(* CoDeSys 2.3 project: cy_64_Desenzano_geolum_1.pro *)
(* Title: cy-wg-24 - ClevergyAS *)
(* Author: Andrea Laini *)
(* Libraries: mod_com.lib 16.5.13 14:00:50, SerComm.lib 16.5.13 14:00:50, GitHubLocalRepository\FIRMWARE_BUILDING_BLOCKS\LuxBlock\LUX_v2.lib 20.4.16 07:33:55, Serial_Interface_01.lib 22.4.13 12:50:14, WagoLibLed.lib 17.6.13 10:40:56, Modb_l05.lib 13.5.15 10:30:08, SysLibFile.lib 16.5.13 14:00:50, Util.lib 16.5.13 14:00:50, GitHubLocalRepository\FIRMWARE_BUILDING_BLOCKS\AstrBlock\obj_ASTR_v2.lib 20.4.16 07:33:55, SYSLIBCALLBACK.LIB 16.5.13 14:00:50, WAGO-CODESYS-LIBS\OSCAT\oscat_basic_333_pfc_2000.lib 10.4.16 18:08:12, SysLibRtc.lib 16.5.13 14:00:50, SysLibSockets.lib 22.5.14 16:16:32, SysLibEvent.lib 16.5.13 14:00:50, SysLibTime.lib 16.5.13 14:00:48, SysLibPlcCtrl.lib 16.5.13 14:00:50, GitHubLocalRepository\FIRMWARE_BUILDING_BLOCKS\CronoBlocks\crono_pfc2000.lib 20.4.16 07:33:55, SysLibStr.lib 16.5.13 14:00:50, Standard.lib 20.5.14 08:13:26, GitHubLocalRepository\FIRMWARE_BUILDING_BLOCKS\01_Lib_ClevergyUtils\ClevergyUtils_pcf2000.lib 20.4.16 07:33:55, Iecsfc.lib 16.5.13 14:00:50 *)

(* PLC configuration (modules and I/O channels)
VPN_STATUS AT %IX0.0 [BOOLOnX_I] I 1: Digital Input
DI02 AT %IX0.1 [BOOLOnX_I] I 2: Digital Input
COORD_STATUS AT %IX0.2 [BOOLOnX_I] I 3: Digital Input
DI04 AT %IX0.3 [BOOLOnX_I] I 4: Digital Input
Modbus variables [PFC200MODBUS] node 1, in %IB0 out %QB0 {PlcStopBehaviour = 1; FiledbusErrorBehaviour = 1; TcpOperation = 0; TcpPort = 502; TcpTimeout = 600; UdpOperation = 0; UdpPort = 502; RtuOperation = 0; NodeId = 200; ResponseTimeout = 5000; Interface = 0; Baud = 38400; StopBits = 2; Parity = 0; FlowCtrl = 0; PhysInterface = 1}
Modbus-Master [MB_MASTER] node 2, in %IB0 out %QB0
*)

(* Global variable list: Global_Constants *)
VAR_GLOBAL CONSTANT

	Plant_NAME			: STRING :='cySN:64  cyVER:0 - Desenzano lab testing';
	Plant_SN				: DWORD  :=64;	  	(* S/N Impianto di telecontrollo *)
	Plant_SW_VER			: WORD   :=0;		(* Versione SW installata *)

	(* Plant-dependent constants *)
	LATITUDE 										: REAL:=45.660772;
	LONGITUDE										: REAL:=9.652021;
	ASTRO_TWILIGHT_MORNING_MODE					: BYTE:=50;
	ASTRO_TWILIGHT_EVENING_MODE					: BYTE:=50;
	COUNTRY_CODE 									: STRING:='IT';
	MAX_LUXNUM										: WORD := 150;
	MAX_GEOLUMENNODES								: WORD :=MAX_LUXNUM;
	MAX_RETRY_NO_FEEDBACK_GEOLUMEN_NODES			: WORD:=5;
	MAX_RETRY_STATUS_NOT_ALIGNED_GEOLUMEN_NODES       : WORD:=60;

	(* Internal, tech const *)
	MAX_ARRAY_MSG	: BYTE:=250;
	ANALOG			: BOOL:=0;
	DIGITAL			: BOOL:=1;

	(* Filesystem *)
	FilesPath  			: STRING :='/media/sd/';
	MapConf_Path			: STRING :=	'/media/sd/';

	Luxlist_FileName	: STRING :='_LUX_LIST.txt';
	Cfg_FileName		: STRING :='CFG.txt';

	(* Colour Visu *)
	COLOR_RED			: DWORD 	:= 16#2020F0;
	COLOR_YELLOW		: DWORD	:= 16#20F0F0;
	COLOR_GREEN		: DWORD	:= 16#20F020;
	COLOR_GREEN_OFF	 : DWORD	:= 16#108010;

	(* TCP Logger *)
	Logger_SERVER		: STRING:='';
	Logger_IP				: STRING:='192.168.100.3';
	Logger_PORT			: WORD  :=80;
	Logger_GETSTART		: STRING:='GET /cygmsrv/hsgm.ashx?';
	Logger_GETEND		: STRING:='$R$N$R$N';
	Logger_CHECK			: STRING:='True';
	Logger_CRLF			: STRING:='$R$N';
	Logger_DataFile		: STRING:='/media/sd/LOG.DAT';
	Logger_DataFileOld	: STRING:='/media/sd/LOG.BCK';
	Logger_IndexFile	: STRING:='/media/sd/LOG.IDX';
	Logger_ConnRetries	: BYTE:=5;
	Logger_RecoverMsgs	: BYTE:=25;

	(* TCP Remote *)
	Remote_PORT			: WORD  :=10;
	Remote_WELCOME		: STRING:='Connected$R$N';
	Remote_OK			: STRING:='OK$R$N';
	Remote_ERROR		: STRING:='ERROR$R$N';

	(* TCP Sockets *)
	MAX_SEND_TCP_SERVER					 : DWORD:=3000;(*60000*)
	MAX_RECEIVE_TCP_SERVER				 : DWORD:=3000;
	MAX_RECEIVE_TCP_SERVER_SOCKET	 	 : DWORD:=1500;
	MAX_SEND_TCP_CLIENT					 : DWORD:=3000;(*15000*)
	MAX_RECEIVE_TCP_CLIENT				 : DWORD:=1500;
	MAX_RECEIVE_TCP_CLIENT_SOCKET		 : DWORD:=1500;
	MAX_RECEIVE_UDP_SERVER				 : INT  :=1472;
	MAX_RECEIVE_UDP_CLIENT				 : INT  :=1472;
	CONNECT_WATCHDOG_TIME				 : TIME :=t#10s;


END_VAR

(* Global variable list: Global_Retain *)
VAR_GLOBAL RETAIN PERSISTENT

	(* valori retain per i LUX objects*)
	GlobalWorkingtime		: ARRAY [1..MAX_LUXNUM] OF DWORD; (* [sec] Internal working time counter *)
	GlobalPowerOnCycles	: ARRAY [1..MAX_LUXNUM] OF WORD;	(*/DWORD;  *) (* Internal counter of power-on cycles *)
	GlobalEnergyCounter	: ARRAY [1..MAX_LUXNUM] OF WORD; (* DWORD;  *) (* [E-1 kWh] Internal energy counter *)
	GlobalEnergyCounter_t 	: ARRAY [1..MAX_LUXNUM] OF DWORD; (* Temporary energy in E-2*Wsec *)

 	(*Tabella della lista dei lux GEOLUMEN costruita sulla base del file di configurazione*)
	TabListLux : ARRAY [1..MAX_LUXNUM] OF type_TabListLuxGeolumen;

	LuxElement		: ARRAY [1..MAX_LUXNUM] OF obj_LUX;  (* Lista di variabili Lux   *)
	LuxGeolumenChangeFlag : ARRAY [1..MAX_LUXNUM] OF INT;

	(*configurazione degli astro *)
	ASTR_CONFIG   : ARRAY [1..MAX_LUXNUM] OF  type_ASTR_config;

	USE_RETAIN:BOOL:=FALSE;

END_VAR

(* Global variable list: Global_Variables *)
VAR_GLOBAL

	SYS    : typ_SYS;
	Logger : typ_Logger;

	LAMP : LAMP_AL_GENERALE;

	PLC_ID				: STRING:='1' ; (* Identificativo del plc - interno al file cfg.txt  *)

	SyncLogRequest: BOOL:=FALSE;
	TimerLogLux : ARRAY[1..15] OF TON;
	TimerLogLuxSync : ARRAY[1..15] OF TON;
	TimerLogLuxSyncDone : ARRAY[1..15] OF BOOL;
	TimingLuxBase : TIME;
	logRowLux:INT:=0;

	TimerLogAstro : ARRAY[1..15] OF TON;
	TimerLogAstroSync : ARRAY[1..15] OF TON;
	TimerLogAstroSyncDone : ARRAY[1..15] OF BOOL;
	TimingAstroBase : TIME;
	tIndex:INT;
	logRowAstro:INT:=0;

	GeolumenNodeList	:GeolumenNodeList;

	(* Astro crono *)
	ASTR   			: ARRAY [1..MAX_LUXNUM] OF obj_ASTR;
	astroGen : obj_ASTR;
	CronEd : obj_CRON_EDITOR:=(crono_type:='ASTR');

	(*Lux *)
	MsgRecBuffer	: ARRAY[0..MAX_ARRAY_MSG ] OF type_MsgReceive; (*Array contenente i messaggi in arrivo e gestito in modo circolare*)
	KEYON :BOOL;

	DataLuxForVis	: ARRAY [1..MAX_LUXNUM] OF type_DataLuxForVis;	(*ARRAY ordinato contenente i valori Status_Vis e del timer utilizzati per la visualizzazione (PLC_Visualization)*)

	LuxGeolumenNodes : ARRAY [1..MAX_LUXNUM] OF obj_GeolumenNode:=(MAX_RETRY_NO_FEEDBACK:=MAX_RETRY_NO_FEEDBACK_GEOLUMEN_NODES,
															MAX_RETRY_STATUS_NOT_ALIGNED:=MAX_RETRY_STATUS_NOT_ALIGNED_GEOLUMEN_NODES);

	LuxGeolumenNodesAlignFlags : ARRAY [1..MAX_LUXNUM] OF BOOL:=FALSE;

	(*Geolumen rs232 dependent*)
	COM0:SERIAL_INTERFACE := (xOPEN_COM_PORT := TRUE, bCOM_PORT_NR  := 0, cbsBYTESIZE := BS_8,
							cbBAUDRATE := BAUD_38400, cpPARITY := PARITY_NO, csSTOPBITS := STOPBITS_1, cfFLOW_CONTROL := NO_FLOW_CONTROL);
	ReceiveBuffer, ReceiveBufferTrash	:typRing_Buffer;
	xCoupledAll		:BOOL;
	obj_GeolumenCoordinator:obj_GeolumenCoordinator;
	LuxGeolumenDiagnostics:LuxGeolumenDiagnostics;
	SendDataQueue:SendDataQueue;

END_VAR

(* Data type in System *)
TYPE en_MsgType :
(
	COMPLETED:=0, (*Il messaggio è stato elaborato*)
	REQAUTH0:= 1,  (*Richiesta in corso a cui rispondere*)
	REQAUTH1:=2,  (*Nodo già acquisito in rete*)
	DATAREC:=3,
	ECHO:=4,
	NODE_DELETED:=5
);
END_TYPE

(* Data type in System *)
TYPE en_StartingState :
(
	NOT_AUTHORISE  := 0,
	READ_NODE
);
END_TYPE

(* Data type *)
TYPE type_ASTR_config :
STRUCT
	id:DWORD;
	twilightMorningMode:BYTE;
	twilightEveningMode:BYTE;
	preSunrise:BYTE;
	postSunrise:BYTE;
	preSunset:BYTE;
	postSunset:BYTE;
END_STRUCT
END_TYPE

(* Data type in DT_LUX_GEOLUMEN *)
TYPE type_LuxGeolumenStatus :
STRUCT
	ID_Geolumen: DWORD;
	DimmValue_0 : WORD;
	DimmValue_1 : WORD;
	DimmValue_2 : WORD;
END_STRUCT
END_TYPE

(* Data type in System *)
TYPE type_MsgReceive :
STRUCT
	Msg		:STRING (255);
	MsgType	: en_MsgType; (*Indica il tipo di messaggio STS0, STS1,...*)
	dwMacAdd	: DWORD;

END_STRUCT
END_TYPE

(* Data type in DT_LUX_GEOLUMEN *)
(* Struttura utile per la lista dei lux *)

TYPE type_TabListLuxGeolumen :
STRUCT
	LuxNumber	: DWORD;
	LuxID_Geolumen		: DWORD;
	MacAdd	: DWORD;
	MacAddH	: WORD;
	MacAddL	: WORD;
	StMacAdd	: STRING(8);
	xCoupled	: BOOL;
END_STRUCT
END_TYPE

(* POU PLC_PRG, ST *)
PROGRAM PLC_PRG
VAR CONSTANT
	TIME_LUX_LOG_NORMAL:TIME:=T#5m;
	TIME_ASTRO_LOG_NORMAL:TIME:=T#6m30s;
END_VAR
VAR

 	Timer1: TON;  (*Fast controls tick *)
  	Timer2: TON; (* Plant control tick *)
	Timer3: TON; (* Logger timer *)
	Timer4: TON; (* Logger timer *)
	Timer5: TON; (* Logger timer *)


	xOpenPort		: BOOL := TRUE;
	xInitPort			: BOOL;
	xSendActive	: BOOL;
	SendString		: STRING(255) := 'CMD_AUTHORISE=1';
	xStartSend		: BOOL;

(* Application vars *)



	i :INT :=0;
	InitCom: BOOL;
	temp 		: BYTE;
	temp2		: INT;



	LuxCount	: WORD;
	LuxEnInfo	: BOOL;
	ValInCrono	: INT; (* Valore del setpoint del crono *)
	counter		: WORD;


	tmpIndex:INT;



END_VAR
(*
	Network setup:
		IP  = 192.168.100.2 | MSK = 255.255.255.0
		GW	= 192.168.100.1 | DNS = 192.168.100.1
		SNTP = 193.204.114.232 (3600s) ==> 192.168.100.3
*)


(*==============================*)
(*=====    Main control machine    ====*)
(*==============================*)

MainCtrl();

Logger_Proc();

Remote_Proc();
END_PROGRAM
ACTION MainCtrl:
CASE Sys.Status OF

	S_STARTUP:
		(* Load the allowed Geolumen nodes *)
		GeolumenNodeList();
		FOR counter := 1 TO MAX_LUXNUM DO
			LuxElement[counter].DimmingType:=1;
			LuxElement[counter].CTRL_MODE := 2 ; (* TabDefaultLux[counter].Mode; //copio il mode nella tabella delle variabili dei lux 	*)
			LuxElement[counter].CTRL_MODE_backUp := 2;  (* TabDefaultLux[counter].Mode; //salvo il mode di backup per il ripristina modo	*)
		END_FOR

		(* apro la porta seriale *)
		xSendActive:=FALSE;
		COM0((*	bCOM_PORT_NR 	:= 0,
				cbBAUDRATE     	 := BAUD_38400,
			(*	cbBAUDRATE 		:= wBaudRate, *)
				cbsBYTESIZE		:= BS_8,  (*bDataBits,*)
				cpPARITY			:= PARITY_NO, (* bParity,*)
				csSTOPBITS		:= STOPBITS_1,
				cfFLOW_CONTROL	:= NO_FLOW_CONTROL,	(*bFlowControl,			*) *)
				utRECEIVE_BUFFER := ReceiveBuffer,
				ptSEND_BUFFER	:= ADR(SendString),
				xINIT				:=  xInitPort,
		     		xOPEN_COM_PORT 	:= TRUE,	(*xOpenPort,*)
				iBYTES_TO_SEND	:= LEN(SendString)+1,
				xSTART_SEND		:= xSendActive );

		IF COM0.xCOM_PORT_IS_OPEN THEN
			Sys.Status:=S_INIT_RTC;
		END_IF

	S_INIT_RTC:

		(* anzitutto blocco auto-accesso da parte dei nodi*)
		obj_GeolumenCoordinator.blockNodeAutoAdd_direct();

		(* Check RTC and update from network *)
		RTC_Update();
		(* Check time *)
		IF Sys.Time_Year>2000 THEN
			obj_GeolumenCoordinator.updateNetworkTime();
			Sys.Status:=S_INIT_VAR;
		END_IF

	S_INIT_VAR:
		(*ripeto il comando di esclusione di accesso da parte dei nodi, per sicurezza*)
		obj_GeolumenCoordinator.blockNodeAutoAdd();

		(* inizializzo gli astro con eventale stato retain *)
		FOR i:=1 TO max_luxnum DO
			ASTR[i].ID:=ASTR_CONFIG[i].ID;
			ASTR[i].rLatitude:=LATITUDE;
			ASTR[i].rLongitude:=LONGITUDE;
			ASTR[i].countryCode:=COUNTRY_CODE;
			IF(USE_RETAIN=FALSE) THEN
				ASTR[i].twilightEveningMode :=ASTRO_TWILIGHT_EVENING_MODE;
				ASTR[i].twilightMorningMode :=ASTRO_TWILIGHT_MORNING_MODE;
				ASTR_CONFIG[i].preSunrise:=ASTR[i].preSunrise;
				ASTR_CONFIG[i].postSunrise:=ASTR[i].postSunrise;
				ASTR_CONFIG[i].preSunset:=ASTR[i].preSunset;
				ASTR_CONFIG[i].postSunset:=ASTR[i].postSunset;
				ASTR_CONFIG[i].twilightEveningMode:=ASTR[i].twilightEveningMode;
				ASTR_CONFIG[i].twilightMorningMode:=ASTR[i].twilightMorningMode;
			ELSE
				ASTR[i].preSunrise:=ASTR_CONFIG[i].preSunrise;
				ASTR[i].postSunrise:=ASTR_CONFIG[i].postSunrise;
				ASTR[i].preSunset:=ASTR_CONFIG[i].preSunset;
				ASTR[i].postSunset:=ASTR_CONFIG[i].postSunset;
				ASTR[i].twilightEveningMode:=ASTR_CONFIG[i].twilightEveningMode;
				ASTR[i].twilightMorningMode:=ASTR_CONFIG[i].twilightMorningMode;
			END_IF

		END_FOR

		(*chiedo agli eventuali nodi geoluem connesso il loro stato già connessi stato *)
		SendDataQueue(pTxData:=ADR(obj_GeolumenCoordinator.getStatusAllFeedback),ReceiveBufferPtr:=ADR(ReceiveBuffer));
		SendDataQueue.addMessage();
		SendDataQueue();

		Sys.Status:=S_STARTER;

	S_STARTER:
		LogEv(EL_Wrn,EO_SYS,0,1,CONCAT('System_startup_v',WORD_TO_STRING(Plant_SW_VER)));
		Sys.Status:=S_RUNNING;

	S_RUNNING:

		astroGen(ID:=1);

		Timer1(IN:=NOT Timer1.Q,PT:=T#50ms);
		IF Timer1.Q THEN
			(* Update meters *)
			SCA_Proc();
			(* Update system checks *)
			SYS_Proc();
		END_IF

		Timer2(IN:=NOT Timer2.Q,PT:=T#500MS);
		IF Timer2.Q THEN
			(* Read current date/time *)
			RTC_Update();
		END_IF

		obj_GeolumenCoordinator(ReceiveBufferPtr:=ADR(ReceiveBuffer),MsgRecBufferPtr:=ADR(MsgRecBuffer));

		(* Execute Cron Editor commands *)
		CronEd();

		(*Timer4(IN:=NOT Timer4.Q,PT:=T#500ms);
		IF Timer4.Q THEN*)



			FOR LuxCount:=1 TO  MAX_LUXNUM DO

				(*eseguo diagnostica lux*)
				LuxGeolumenDiagnostics();

				IF  LuxElement[LuxCount].ID <> 0  THEN (* esegue scansione dei lux dell'impianto solo se presenti *)

					(* salvo lo stato desiderato corrente del LuxGeolumenNode *)
					LuxGeolumenChangeFlag[LuxCount]:=LuxGeolumenNodes[LuxCount].desideredDimmValue;

					CASE LuxElement[LuxCount].CTRL_MODE OF
						(*
						0:
						1:	 *)
						2:

							IF  ASTR[LuxCount].ID <> 0 THEN
								(* se il mode è settato come cronografo gestisco accensione a orologio *)
								ASTR[LuxCount]( localTime:=Sys.Time_CT_DT,SetPoint=>ValInCrono);
								LuxElement[LuxCount].ValInCronoInLux:=ValInCrono;
							END_IF

					END_CASE

					LuxElement[LuxCount](	LuxAnalogOut => LuxGeolumenNodes[LuxCount].desideredDimmValue,
										WorkingTime:=GlobalWorkingtime[LuxCount],
										PowerOnCycles:=GlobalPowerOnCycles[LuxCount],
										EnergyCounter:=GlobalEnergyCounter[LuxCount],
										EnergyCounter_t:=GlobalEnergyCounter_t[LuxCount],KeyQty:=2);  (*, KeyMode:=KeyTest.KeyMode); *)

					(* aggiorno lo stato desiderato del LUX GeolumenNode*)
					LuxGeolumenNodes[LuxCount].updateDesideredState();
					(* se è diverso dal precedente, invio richiesta modifica stato *)
					IF(LuxGeolumenChangeFlag[LuxCount]<>LuxGeolumenNodes[LuxCount].desideredDimmValue) THEN
						(*invio set*)
						SendDataQueue(pTxData:=ADR(LuxGeolumenNodes[LuxCount].toSendSetString),ReceiveBufferPtr:=ADR(ReceiveBuffer));
						SendDataQueue.addMessage();
						(*invio get*)
						SendDataQueue(pTxData:=ADR(LuxGeolumenNodes[LuxCount].toSendGetString),ReceiveBufferPtr:=ADR(ReceiveBuffer));
						SendDataQueue.addMessage();
						SendDataQueue();
					END_IF

					LuxGeolumenNodes[LuxCount].checkStatusANDPresence();
					LuxGeolumenNodesAlignFlags[LuxCount]:=isGeolumenIEqualStatus(LuxGeolumenNodes[LuxCount].desideredState, LuxGeolumenNodes[LuxCount].feedbackState);

				END_IF
			END_FOR
		(*END_IF*)

		(* elaboro comunque coda messaggi in uscita e ingresso*)
		SendDataQueue(ReceiveBufferPtr:=ADR(ReceiveBuffer));


		(*Timer3(IN:=NOT Timer3.Q,PT:=T#5m);
		IF Timer3.Q THEN
			(* Trig logger *)
			LogTrig();
		END_IF*)

		IF SyncLogRequest = FALSE THEN

			timingLuxBase:=TIME_LUX_LOG_NORMAL;
			timingAstroBase:=TIME_ASTRO_LOG_NORMAL;

			FOR tIndex:=1 TO 15 DO
				TimerLogLux[tIndex](IN:=NOT TimerLogLux[tIndex].Q,PT:=timingLuxBase+INT_TO_TIME(TIME_TO_INT(t#5s)*tIndex));
					IF TimerLogLux[tIndex].Q THEN
						(* Trig logger *)
						objLuxLog(tIndex);
					END_IF
			END_FOR

			FOR tIndex:=1 TO 15 DO
				TimerLogAstro[tIndex](IN:=NOT TimerLogAstro[tIndex].Q,PT:=timingAstroBase+INT_TO_TIME(TIME_TO_INT(t#5s)*tIndex));
				IF TimerLogAstro[tIndex].Q THEN
					(* Trig logger *)
					objAstroLog(tIndex);
				END_IF
			END_FOR

		ELSE

			IF logRowLux <15 THEN
			FOR tIndex:=1 TO 15 DO
				TimerLogLuxSync[tIndex](IN:=NOT TimerLogLuxSync[tIndex].Q,PT:=timingLuxBase+INT_TO_TIME(TIME_TO_INT(t#5s)*tIndex));
					IF TimerLogLuxSync[tIndex].Q AND TimerLogLuxSyncDone[tIndex] = FALSE THEN
						(* Trig logger *)
						objLuxLog(tIndex);
						logRowLux:=(logRowLux+1) MOD 16 + logRowLux/16;
						TimerLogLuxSyncDone[tIndex]:=TRUE;
					END_IF
			END_FOR
			END_IF

			IF logRowAstro <15 THEN
			FOR tIndex:=1 TO 15 DO

				TimerLogAstroSync[tIndex](IN:=NOT TimerLogAstroSync[tIndex].Q,PT:=timingAstroBase+INT_TO_TIME(TIME_TO_INT(t#5s)*tIndex));
				IF TimerLogAstroSync[tIndex].Q AND TimerLogAstroSyncDone[tIndex] = FALSE THEN
					(* Trig logger *)
					objAstroLog(tIndex);
					logRowAstro:=(logRowAstro+1) MOD 16  +logRowLux/16;
					TimerLogAstroSyncDone[tIndex] :=TRUE;
				END_IF
			END_FOR
			END_IF

			IF logRowAstro>=15 AND logRowLux>=15 THEN SyncLogRequest:=FALSE; END_IF

		END_IF



	S_RELOAD:

		(*ricaricamento file di configurazione: azzero tutti i Lux, Astr GeolumenNodes e ricomincio da capo *)
		LogEv(EL_Wrn,EO_SYS,0,1,CONCAT('System_reload_config_file',WORD_TO_STRING(Plant_SW_VER)));
		FOR counter := 1 TO MAX_LUXNUM DO
			TabListLux[counter].LuxID_Geolumen:=0;
			TabListLux[counter].MacAdd:=0;
			TabListLux[counter].MacAddH:=0;
			TabListLux[counter].MacAddL:=0;
			TabListLux[counter].StMacAdd:='';
			TabListLux[counter].LuxNumber:=0;
			TabListLux[counter].xCoupled:=FALSE;
			LuxElement[counter].ID:=0;
			ASTR[counter].ID:=0;
			LuxGeolumenNodes[counter].ID_Lux:=0;
			LuxGeolumenNodes[counter].ID_Geolumen:=0;
		END_FOR
		FOR counter := 0 TO MAX_ARRAY_MSG  DO
				MsgRecBuffer[i].Msg:='';
				MsgRecBuffer[i].MsgType := COMPLETED;
				MsgRecBuffer[i].dwMacAdd:=0;
		END_FOR
		xCoupledAll:=FALSE;

		Sys.Status:=S_STARTUP;

ELSE
	Sys.Status:=S_STARTUP;
END_CASE;
END_ACTION

(* POU TCP_Remote/Remote_Proc, ST *)
PROGRAM Remote_Proc
VAR
	s1:         	TCPSERVER;
	Enable: 		BOOL;
	Connected: 		BOOL;
	Error: 			DINT;

	TxData:			ARRAY [0..MAX_SEND_TCP_SERVER] OF BYTE;
	TxLen:			DINT;
	TxTrig:			BOOL;

	RxData:			ARRAY [0..MAX_RECEIVE_TCP_SERVER] OF BYTE;
	RxLen:			DINT;

	Status:			DINT;

	(* Command interpreter *)

	Cmd_Buf:		ARRAY [0..MAX_RECEIVE_TCP_SERVER] OF BYTE;
	Cmd_Buf_U16:	POINTER TO WORD;
	Cmd_Buf_INT:	POINTER TO INT;
	Cmd_BufLen:		WORD;
	Cmd_St:			WORD;

	Cmd_Obj:		WORD;
	Cmd_ObjIdx:		WORD;
	Cmd_ObjIdx_Low:		BYTE;
	Cmd_ObjIdx_High:		BYTE;
	Cmd_C:			WORD;
	Cmd_R:			WORD;
	Cmd_CLen:		WORD;
	Cmd_RLen:		WORD;

	i : WORD;
	j : INT;
	s2 : STRING;

	(* per aggiornare la data e l'ora *)
	SetAnno: INT;
	SetMese: INT;
	SetGiorno: INT;
	SetOra: INT;
	SetMinuti: INT;
	SetSecondi: INT;

	Plant_SW_VER: BOOL;
         (* specific for lux *)
	x: INT;
	NewValueTimer : DWORD;

	ASTR_ARRAY: BOOL;
END_VAR
(*=== State machine ===*)
CASE Status OF
	0: (* Startup *)
		TxLen:=0; TxTrig:=FALSE;
		RxLen:=0;
		Enable:=TRUE;
		Status:=1;

	1: (* Wait incoming connection *)
		IF Connected THEN
			(* Log access *)(*
			LogEv(EL_Log,EO_VPN,1,5,'Remote');*)
			(* Send welcome message *)(*
			ADDSTRING(pTxData:=ADR(TxData), pString:=ADR(Remote_WELCOME), TxLen:=TxLen);
			TxTrig:=TRUE;*)
			(* Reset vars *)
			Cmd_BufLen:=0;
			Cmd_St:=0;
			Status:=2;
		END_IF
		IF Error>1 THEN
			Enable:=FALSE;
			Status:=0;
		END_IF

	2: (* Wait command *)
		IF RxLen>0 THEN
			(*=== Interpreter start ===*)
			IF Cmd_BufLen+(RxLen/2)>=MAX_RECEIVE_TCP_SERVER THEN
				(* ERROR *)
				Cmd_BufLen:=0;
			ELSE
				i:=HEXTORAW(pString:=ADR(RxData), StringLen:=DINT_TO_WORD(RxLen), pData:=ADR(Cmd_Buf[Cmd_BufLen]));
				Cmd_BufLen:=Cmd_BufLen+i;
			END_IF
			IF Cmd_BufLen>=8 THEN
				Cmd_Buf_U16:=ADR(Cmd_Buf[6]);
				IF Cmd_BufLen>=(8+Cmd_Buf_U16^) THEN
					Cmd_CLen:=Cmd_Buf_U16^;
					Cmd_Buf_U16:=ADR(Cmd_Buf[0]); Cmd_Obj:=Cmd_Buf_U16^;
					Cmd_Buf_U16:=ADR(Cmd_Buf[2]); Cmd_ObjIdx:=Cmd_Buf_U16^;Cmd_ObjIdx_Low:=Cmd_Buf[2];Cmd_ObjIdx_High:=Cmd_Buf[3];
						(*fix per id maggiori di 255*)
						(*IF Cmd_Buf[3] <>0 THEN
							Cmd_ObjIdx:=ROL(Cmd_ObjIdx,8);
						END_IF*)
					Cmd_Buf_U16:=ADR(Cmd_Buf[4]); Cmd_C:=Cmd_Buf_U16^;
					(* Log command *)(*
					s2:='RCmd_';		s2:=CONCAT(s2,WORD_TO_STRING(Cmd_Obj));
					s2:=CONCAT(s2,'_'); s2:=CONCAT(s2,WORD_TO_STRING(Cmd_ObjIdx));
					s2:=CONCAT(s2,'_'); s2:=CONCAT(s2,WORD_TO_STRING(Cmd_C));
					s2:=CONCAT(s2,'_');	s2:=CONCAT(s2,WORD_TO_STRING(Cmd_CLen));
					LogEv(EL_Log,EO_VPN,1,6,s2);*)
					(* Execute command *)
					Command();
					Cmd_BufLen:=0;
				END_IF
			END_IF
			(*=== Interpreter end ===*)
			RxLen:=0;
		END_IF
		IF NOT Connected THEN
			Status:=0;
		END_IF

ELSE
	Status:=0;
END_CASE


(*=== Execute server lib ===*)
s1(
	xEnable				:= Enable,
	wPortNumber			:= Remote_PORT,
	tServerTimeOut		:= t#15m,
	ptSendData			:= ADR(TxData),
	diSendCount			:= TxLen,
	xStartSend			:= TxTrig,
	aReceiveBuffer		:= RxData,
	diReceiveCount		:= RxLen,
	xClientConnected	=> Connected,
	diError				=> Error
);
END_PROGRAM
ACTION Cmd_ASTR:
(* Check index *)
IF Cmd_ObjIdx < 1 THEN
	Cmd_R := 2; (* //id del lux fuori range*)
	RETURN ;
END_IF

x := 1 ;
WHILE ( x <=MAX_LUXNUM ) AND ( Cmd_ObjIdx <>  ASTR[ x ] . ID )  DO
	x := x + 1 ;
END_WHILE

(*
	Cmd_ObjIdx => logical id for Clevergy
	x=> where the object of ID Cmd_ObjIdx is placed inside the internal array
*)
IF  x <=MAX_LUXNUM AND Cmd_ObjIdx =  ASTR [ x ] . ID THEN

(* Process command *)
CASE Cmd_C OF

	1: (* GET PROFILE *)
		IF Cmd_CLen<>3 THEN
			Cmd_R:=4;
		ELSE
			(* Load profile *)
			CronEd.CN_Sel:=WORD_TO_BYTE(Cmd_ObjIdx);
			Cmd_Buf_U16:=ADR(Cmd_Buf[8]);
			CronEd.CN_YSel:=Cmd_Buf_U16^;
			CronEd.PR_Sel:=Cmd_Buf[10];
			CronEd.PR_Load_Exe();
			(* Copy data *)
			Cmd_RLen:=192;
			TxLen:=TxLen+RAWTOHEX(ADR(CronEd.PR.Setpoint),192,ADR(TxData[TxLen]));

		END_IF

	2: (* SET PROFILE *)
		IF Cmd_CLen<>(3+192) THEN
			Cmd_R:=4;
		ELSE
			(* Save profile *)
			CronEd.CN_Sel:=WORD_TO_BYTE(Cmd_ObjIdx);
			Cmd_Buf_U16:=ADR(Cmd_Buf[8]);
			CronEd.CN_YSel:=Cmd_Buf_U16^;
			CronEd.PR_Sel:=Cmd_Buf[10];
			MEMCPY(ADR(Cmd_Buf[11]),ADR(CronEd.PR.Setpoint),192);
			CronEd.PR_Save_Exe();

			ASTR[x].restartInternalCrono();
		END_IF

	5: (* GET CALENDAR MONTH *)
		IF Cmd_CLen<>3 THEN
			Cmd_R:=4;
		ELSE
			(* Load calendar *)
			CronEd.CN_Sel:=WORD_TO_BYTE(Cmd_ObjIdx);
			Cmd_Buf_U16:=ADR(Cmd_Buf[8]);
			CronEd.CN_YSel:=Cmd_Buf_U16^;
			CronEd.CA_Sel:=Cmd_Buf[10];
			CronEd.CA_Load_Exe();
			(* Copy data *)
			Cmd_RLen:=32;
			TxLen:=TxLen+RAWTOHEX(ADR(CronEd.CA.Profile),32,ADR(TxData[TxLen]));
		END_IF

	6: (* SET CALENDAR MONTH *)
		IF Cmd_CLen<>(3+32) THEN
			Cmd_R:=4;
		ELSE
			(* Save calendar *)
			CronEd.CN_Sel:=WORD_TO_BYTE(Cmd_ObjIdx);
			Cmd_Buf_U16:=ADR(Cmd_Buf[8]);
			CronEd.CN_YSel:=Cmd_Buf_U16^;
			CronEd.CA_Sel:=Cmd_Buf[10];
			MEMCPY(ADR(Cmd_Buf[11]),ADR(CronEd.CA.Profile),32);
			CronEd.CA_Save_Exe();
		END_IF

	9: (* CRON RESTART *)
		ASTR[x].restartInternalCrono();

	10: (* GET ASTR PARAMETERS *)


		Cmd_RLen:=10;
		TxLen:=TxLen + RAWTOHEX_BYTE(ADR(TxData[TxLen]),ASTR[x].preSunrise);
		TxLen:=TxLen + RAWTOHEX_BYTE(ADR(TxData[TxLen]),ASTR[x].postSunrise);
		TxLen:=TxLen + RAWTOHEX_BYTE(ADR(TxData[TxLen]),ASTR[x].preSunset);
		TxLen:=TxLen + RAWTOHEX_BYTE(ADR(TxData[TxLen]),ASTR[x].postSunset);
		TxLen:=TxLen + RAWTOHEX_BYTE(ADR(TxData[TxLen]),ASTR[x].twilightEveningMode);
		TxLen:=TxLen + RAWTOHEX_BYTE(ADR(TxData[TxLen]),ASTR[x].twilightMorningMode);



	11: (* SET ASTR PARAMETERS *)
		IF Cmd_CLen<>(12/2) THEN
			Cmd_R:=4;
		ELSE

			ASTR[x].preSunrise:=Cmd_Buf[8];
			ASTR[x].postSunrise:=Cmd_Buf[9];
			ASTR[x].preSunset:=Cmd_Buf[10];
			ASTR[x].postSunset:=Cmd_Buf[11];
			ASTR[x].twilightEveningMode:=Cmd_Buf[12];
			ASTR[x].twilightMorningMode:=Cmd_Buf[13];


			ASTR_CONFIG[x].preSunrise:=ASTR[x].preSunrise;
			ASTR_CONFIG[x].postSunrise:=ASTR[x].postSunrise;
			ASTR_CONFIG[x].preSunset:=ASTR[x].preSunset;
			ASTR_CONFIG[x].postSunset:=ASTR[x].postSunset;
			ASTR_CONFIG[x].twilightEveningMode:=ASTR[x].twilightEveningMode;
			ASTR_CONFIG[x].twilightMorningMode:=ASTR[x].twilightMorningMode;
			USE_RETAIN:=TRUE;

		END_IF

ELSE
	Cmd_R:=3;
END_CASE

ELSE
	Cmd_R := 2 ; (*//id del lux non presente in lista*)
END_IF
END_ACTION
ACTION Cmd_LUX:
(* Check index *)
IF Cmd_ObjIdx < 1 THEN
	Cmd_R := 2; (* //id del lux fuori range*)
	RETURN ;
END_IF

x := 1 ;
WHILE ( x <=MAX_LUXNUM ) AND ( Cmd_ObjIdx <>  LuxElement [ x ] . ID )  DO
	x := x + 1 ;
END_WHILE

IF  x <=MAX_LUXNUM AND  Cmd_ObjIdx =  LuxElement [ x ] . ID THEN

	(* Process command *)
 	CASE Cmd_C OF

		0 : (* Restore default functioning mode *)
			LuxElement [ x ] . CTRL_MODE := LuxElement [ x ] . CTRL_MODE_backUp ;
			LuxElement [ x ] (     WORKINGTIME := GlobalWorkingTime [ x ] ,
							POWERONCYCLES :=
							GlobalPowerOnCycles [ x ] ,
							ENERGYCOUNTER := GlobalEnergyCounter [ x ] ,
							ENERGYCOUNTER_T :=
							GlobalEnergyCounter_t [ x ] ,
							CtrlExton := KEYON ) ;

		1 : (* Reset statistic counter *)
			LuxElement [ x ] . StatReset (  WORKINGTIME := GlobalWorkingTime [ x ] ,
									POWERONCYCLES := GlobalPowerOnCycles [ x ] ,
									ENERGYCOUNTER :=GlobalEnergyCounter [ x ] ,
									ENERGYCOUNTER_T:= GlobalEnergyCounter_t [ x ] ,
									CtrlExton :=KEYON ) ;

		2 , 3 : (* Switch On (command=2) or Off (command=3) lux *)
			CASE Cmd_C OF
				2 : (*switch a Manuale ON*)
					LuxElement [ x ] . CTRL_MODE := 1 ; (*// Set to manuale ON *)
					LuxElement [ x ].DimmingValForManual:=LuxElement [ x ].MAX_DIMM_VALUE;
					LuxElement [ x ] (     WORKINGTIME := GlobalWorkingTime [ x ] ,
									POWERONCYCLES:= GlobalPowerOnCycles [ x ] ,
									ENERGYCOUNTER :=GlobalEnergyCounter [ x ] ,
									ENERGYCOUNTER_T :=GlobalEnergyCounter_t [ x ] ,
									CtrlExton := KEYON ) ;

				3 : (*switch a Manuale OFF*)
					LuxElement [ x ] . CTRL_MODE := 0 ; (*// Set to manuale OFF *)
					LuxElement [ x ].DimmingValForManual:=0;
					LuxElement [ x ] (     WORKINGTIME := GlobalWorkingTime [ x ] ,
									POWERONCYCLES:= GlobalPowerOnCycles [ x ] ,
									ENERGYCOUNTER :=GlobalEnergyCounter [ x ] ,
									ENERGYCOUNTER_T :=GlobalEnergyCounter_t [ x ] ,
									CtrlExton := KEYON ) ;

			END_CASE

		4 : (* Modify timer value *)
			IF  LuxElement [ x ] . CTRL_Mode = 03 THEN
				(*la modifica ha senso per i lux a timer*)
				NewValueTimer := BYTE_TO_DWORD ( Cmd_Buf [ 8 ] ) ;
				NewValueTimer := SHL ( NewValueTimer , 8 ) ;	
				NewValueTimer := NewValueTimer + BYTE_TO_DWORD ( Cmd_Buf [ 9 ] ) ;
				NewValueTimer := SHL ( NewValueTimer , 8 ) ;
				NewValueTimer := NewValueTimer + BYTE_TO_DWORD ( Cmd_Buf [ 10 ] ) ;
				NewValueTimer := SHL ( NewValueTimer , 8 ) ;
				NewValueTimer := NewValueTimer + BYTE_TO_DWORD ( Cmd_Buf [ 11 ] ) ;
				(*TabLuxPsg [ x ] . TimerOn := DWORD_TO_TIME ( NewValueTimer *1000 ) ;*) (*REMOVE THIS LINE *)

				FOR x := 1 TO MAX_LUXNUM DO
					IF LuxElement [ x ] . ID = Cmd_ObjIdx THEN
						LuxElement [ x ] . LuxTimer := DWORD_TO_TIME (NewValueTimer * 1000 ) ; (*//set del nuovo valore del timer del lux*)
					END_IF
				END_FOR
			ELSE
				Cmd_R := 3 ; (*//Comando errato / non previsto*)
			END_IF
		(* 5: (* Modify dimming value for timer control *) *)
		(* 6: (* Modify dimming value for key control *) *)

		(* 7: (* Modify start and stop orari di funzionamento dei lux a timer *) *)

	8: (* SET MANUAL DIMMLEVEL*)
		IF Cmd_CLen<>(1) THEN
			Cmd_R:=4;
		ELSE
				IF(Cmd_Buf[8]>0) THEN
					LuxElement [x] . CTRL_MODE := 1 ; (*// Set to manuale on con dimm*)
					LuxElement [x].DimmingValForManual:=Cmd_Buf[8];
				ELSE
					LuxElement [x] . CTRL_MODE := 0 ; (*// Set to manuale off*)
					LuxElement [x].DimmingValForManual:=0;
				END_IF
				LuxElement [x] (    WORKINGTIME := GlobalWorkingTime [x ] ,
				POWERONCYCLES:= GlobalPowerOnCycles [x] ,
				ENERGYCOUNTER :=GlobalEnergyCounter [x] ,
				ENERGYCOUNTER_T :=GlobalEnergyCounter_t [x ] ,
									CtrlExton := KEYON ) ;
		END_IF
		ELSE
			Cmd_R := 3 ; (*//Comando errato / non previsto*)
		END_CASE
ELSE
	Cmd_R := 2 ; (*//id del lux non presente in lista*)
END_IF
END_ACTION
ACTION Cmd_SYS:
(* Check index *)
IF Cmd_ObjIdx<>0 THEN
	Cmd_R:=2;
	RETURN;
END_IF

(* Process command *)
CASE Cmd_C OF

	0: (* ECHO *)
		IF Cmd_CLen<>0 THEN
			TxLen:=0;
		END_IF

	1: (* LOG REQUEST *)
		LogTrig();

	2: (* REARM *)
		Sys.Warning:=FALSE;
		Sys.Alarm:=FALSE;
		Sys.AlarmStop:=FALSE;

	3: (* GET INFO1 *)
		Cmd_RLen:=6;
		TxLen:=TxLen+RAWTOHEX(ADR(Plant_SN),4,ADR(TxData[TxLen]));
		TxLen:=TxLen+RAWTOHEX(ADR(Plant_SW_VER),2,ADR(TxData[TxLen]));

	14: (*  Imposto data e ora del PLC  *)


			Cmd_Buf_U16:=ADR(Cmd_Buf[8]);
			SetAnno:= Cmd_Buf_U16^; 												(* Anno *)
			Cmd_Buf_U16:=ADR(Cmd_Buf[10]);
			SetMese:= Cmd_Buf_U16^;												 	(* mese *)
			Cmd_Buf_U16:=ADR(Cmd_Buf[12]);
			SetGiorno:=( Cmd_Buf_U16^);											 	(* Giorno *)
			Cmd_Buf_U16:=ADR(Cmd_Buf[14]);
			SetOra:=( Cmd_Buf_U16^); 												(* ora *)
			Cmd_Buf_U16:=ADR(Cmd_Buf[16]);
			SetMinuti:= ( Cmd_Buf_U16^);										 	(* Minuti *)
			Cmd_Buf_U16:=ADR(Cmd_Buf[18]);
			SetSecondi:= ( Cmd_Buf_U16^);										 	(* secondi *)

			SysRtcSetTime((SetDataTime(SetAnno,SetMese,SetGiorno,SetOra,SetMinuti,SetSecondi)));

ELSE
	Cmd_R:=3;
END_CASE
END_ACTION
ACTION Command:
(* Default response OK/NODATA *)
Cmd_R:=0;
Cmd_RLen:=0;
TxLen:=16;

(* Check object *)
CASE Cmd_Obj OF

	EO_SYS:
		Cmd_SYS();

	EO_LUX:
		Cmd_LUX();

	EO_ASTR:
		Cmd_ASTR();

ELSE
	Cmd_R:=3;
END_CASE

(* Generate response *)
IF TxLen>0 THEN
	RAWTOHEX(ADR(Cmd_Obj)	,2,ADR(TxData[ 0]));
	RAWTOHEX(ADR(Cmd_ObjIdx),2,ADR(TxData[ 4]));
	RAWTOHEX(ADR(Cmd_R)		,2,ADR(TxData[ 8]));
	RAWTOHEX(ADR(Cmd_RLen)	,2,ADR(TxData[12]));
	TxTrig:=TRUE;
END_IF
END_ACTION

(* POU GeoLumenWrapping/obj_GeolumenCoordinator, ST *)
FUNCTION_BLOCK obj_GeolumenCoordinator
VAR CONSTANT
	getStatusAllFeedback:STRING:='NWK_GET_STATUS$R$N';
END_VAR
VAR_INPUT
	ReceiveBufferPtr : POINTER TO typRing_Buffer;
	MsgRecBufferPtr : POINTER TO ARRAY[0..MAX_ARRAY_MSG ] OF type_MsgReceive;
END_VAR
VAR_OUTPUT
	LastMessage: STRING(255) := '';
END_VAR
VAR

	xOpenPort		: BOOL := TRUE;
	xInitPort			: BOOL;
	xSendActive	: BOOL;
	xStartSend		: BOOL;
	SendString : STRING(255):='';
	pReceiveStr 	: POINTER TO STRING(255);
	StringaDaSeriale 	: STRING(255):='';
	tempStringa : STRING(255) := '';
	ArrayPos		: BYTE;
	LenghtStr	: INT;
	TrimStr1, TrimStr2,TrimNMEAS	: STRING(10);
	contFrame : INT :=0;
	StringCmp1, StringCmp2	: DINT;
	i :INT :=0;
	tempEnd: INT;
	tempBegin: INT;
	tempBegin0: INT;
	InitCom: BOOL;
	temp 		: BYTE;
	temp2		: INT;
	MyString	: STRING(255);
	pString1, pString2	: POINTER TO STRING(255);
	superatoTEMPSTRINGA:STRING(255):='';
	superatoSTRINGADASERIALE:STRING(255):='';
	tmpIndex:INT;
	maxStringaDaSerialeLength:INT:=0;
	maxConcat:INT:=0;
	x	: WORD;
	MacStr	: STRING (8);
	StrToSend	:STRING(50);
	counter, index	: WORD;
	StrLoc			: BYTE;
	StrSaveMacAdd	: STRING;
	StrSaveID		: STRING;
	Str				: STRING;
END_VAR
VAR CONSTANT
	ID_NODE_PREFIX:STRING:='IDN';
	PW0_PREFIX:STRING:='PW0';
	PW1_PREFIX:STRING:='PW1';
	PW2_PREFIX:STRING:='PW2';
	FIELD_SEPARATOR:STRING:=';';
END_VAR
VAR_INPUT
	statusNodeMessage : STRING(255);
END_VAR
VAR_OUTPUT
	idNode : WORD;
	state: TYPE_LuxGeolumenStatus;
END_VAR
VAR
	pwm0 : WORD;
	pwm1 : WORD;
	pwm2 : WORD;
	idNodeStart:INT;
	partialStringNode, partialStringPW0,partialStringPW1,partialStringPW2:STRING;
	posSeparator:WORD;
	idPw0Start:INT;
	idPw1Start:INT;
	idPw2Start:INT;

END_VAR
VAR

	StrMin			: STRING(4);
	StrHour			: STRING(4);
	StartingState	: en_StartingState;
END_VAR
getAndParseMessage();
IF NOT (xCoupledAll) THEN (* Se non tutti i nodi sono accoppiati spedisco autorizzazione a chi ne fa richiesta e fa parte dell'elenco iniziale *)
	SendAuth();
END_IF
ReadID(); (*esegue associazione ID --> Mac Address e lo scrive nella struttura TabListLux *)
AllCoupled(); (* verifica se tutti i Mac Address sono acciopiati con l'ID*)
END_FUNCTION_BLOCK
ACTION AllCoupled:
counter :=1;
xCoupledAll:=FALSE;
WHILE (counter<=MAX_GEOLUMENNODES) DO
	IF TabListLux[counter].xCoupled = FALSE THEN
		RETURN;
	END_IF
	counter:=counter+1;
END_WHILE
IF counter = MAX_GEOLUMENNODES+1 THEN
	xCoupledAll:=TRUE;
END_IF
END_ACTION
ACTION blockNodeAutoAdd:
SendString := 'CMD_AUTHORISE=0$R$N';
SendDataQueue(pTxData:=ADR(SendString),ReceiveBufferPtr:=ADR(ReceiveBuffer));
SendDataQueue.addMessage();
SendDataQueue();
END_ACTION
ACTION blockNodeAutoAdd_direct:
(* Comando di esclusione di accesso da parte dei nodi*)
SendString := 'CMD_AUTHORISE=0$R$N';
SendData(pTxData:=ADR(SendString));
END_ACTION
ACTION GetAndParseMessage:
	xStartSend:=FALSE;
	COM0(	utRECEIVE_BUFFER := ReceiveBufferPtr^,
				ptSEND_BUFFER	:= ADR(SendString),
				xINIT				:=  xInitPort,
		     		xOPEN_COM_PORT 	:= TRUE,
				iBYTES_TO_SEND	:= LEN(SendString)+1,
				xSTART_SEND		:= xStartSend );

		IF pReceiveStr = 0 THEN
			pReceiveStr := ADR(ReceiveBufferPtr^.Data);
		END_IF;

		IF (ReceiveBufferPtr^.Index > 0 ) THEN
			StringaDaSeriale :=  pReceiveStr^ ;
			IF LEN(StringaDaSeriale) > maxStringaDaSerialeLength THEN maxStringaDaSerialeLength:=LEN(StringaDaSeriale); END_IF
			IF(LEN(tempStringa)+LEN(StringaDaSeriale)<=255) THEN
				tempStringa :=CONCAT(tempStringa, StringaDaSeriale);
			ELSE

				tempStringa:='';
				tempStringa :=CONCAT(tempStringa, StringaDaSeriale);
				superatoTEMPSTRINGA:=tempStringa;
				superatoSTRINGADASERIALE:=StringaDaSeriale;
			END_IF
			IF LEN(tempStringa)+LEN(StringaDaSeriale)>maxConcat THEN maxConcat:=LEN(tempStringa)+LEN(StringaDaSeriale); END_IF
			tempBegin:=FIND(tempStringa,'$R$N');
			IF(tempBegin>0) THEN
				LastMessage:=LEFT(tempStringa,tempBegin-1);
				tempStringa:='';

(*				TempStr:=LEFT(LastMessage, 80); *)

				pString2:=ADR(LastMessage);
				pString1:=ADR(MsgRecBuffer[ArrayPos].Msg);

				pString1^:=pString2^;
				LenghtStr:= LEN(MsgRecBuffer[ArrayPos].Msg);
				TrimStr1:=MID(MsgRecBuffer[ArrayPos].Msg, 3, 1); (*Isolo la sottostringa iniziale -  '#!#' *)
				IF(SysStrCmp(TrimStr1, '#.#') = 0) THEN
					TrimStr1:=MID(MsgRecBuffer[ArrayPos].Msg, 7, 4); (*Isolo la sottostringa iniziale - REQAUTH*)
					TrimStr2:=MID(MsgRecBuffer[ArrayPos].Msg, 4, 32); (*Isolo la sottostringa finale - STS0*)
(*					StringCmp1:=SysStrCmp(TrimStr1, 'REQAUTH');  Verifica se sottostringa iniziale = REQAUTH*)
(*					StringCmp2:=SysStrCmp(TrimStr2, 'STS0');  Verifica se sottostringa finale = STS0*)
					IF (SysStrCmp(TrimStr1, 'REQAUTH') = 0 AND SysStrCmp(TrimStr2, 'STS0') = 0) THEN
						MsgRecBuffer[ArrayPos].MsgType := REQAUTH0;
					ELSE
						TrimNMEAS:=MID(MsgRecBuffer[ArrayPos].Msg, 5, 4); (* Isolo la sottostringa iniziale - NMEAS*)
						IF (SysStrCmp(TrimNMEAS, 'NMEAS') = 0  AND   FIND(MsgRecBuffer[ArrayPos].Msg,  '#!#' ) > 0) THEN
							MsgRecBufferPtr^[ArrayPos].MsgType := DATAREC;
							(*identifco a quale nodo lux geolumen si riferisce *)
							parseNodeStatus(statusNodeMessage:=MsgRecBufferPtr^[ArrayPos].Msg);
							IF idNode>=1 AND idNode<=MAX_LUXNUM THEN
								tmpIndex:=getGeolumenNodeByGeolumenId (idNode);
								IF(tmpIndex>0) THEN LuxGeolumenNodes[tmpIndex](feedbackState:=state); LuxGeolumenNodes[tmpIndex].updateFeedbackState(); END_IF
							END_IF
						END_IF
					END_IF
				ELSIF  FIND(MsgRecBufferPtr^[ArrayPos].Msg,  '>' ) = 1 (* Isolo la sottostringa iniziale - > *) THEN
						MsgRecBufferPtr^[ArrayPos].MsgType := ECHO;
				ELSIF  FIND(MsgRecBufferPtr^[ArrayPos].Msg,  'Delete Operation Complete' ) = 1 (* Isolo la sottostringa iniziale - Delete Operation Complete *) THEN
						MsgRecBufferPtr^[ArrayPos].MsgType := NODE_DELETED;
				END_IF


				IF ArrayPos<MAX_ARRAY_MSG+1 THEN
					ArrayPos:=ArrayPos+1;
				ELSE
					ArrayPos:=0;
				END_IF
				MsgRecBufferPtr^[ArrayPos].Msg:='';
				MsgRecBufferPtr^[ArrayPos].MsgType := COMPLETED;
				MsgRecBufferPtr^[ArrayPos].dwMacAdd:=0;
				MsgRecBufferPtr^[ArrayPos+1].Msg:='';
				MsgRecBufferPtr^[ArrayPos+1].MsgType := COMPLETED;
				MsgRecBufferPtr^[ArrayPos+1].dwMacAdd:=0;
		END_IF;

		    (* clean buffer *)
		    ReceiveBufferPtr^.Index := 0;
		    FOR i:=0 TO 255 DO
		       ReceiveBufferPtr^.Data[i]:=16#00;
		    END_FOR;

		    (* conto i frame che ho ricevuto *)
		    contFrame:=contFrame+1;

		END_IF;
END_ACTION
ACTION parseNodeStatus:
(*get node id - idn*)
idNodeStart:=FINDP(statusNodeMessage,ID_NODE_PREFIX,1);
partialStringNode:=DELETE(statusNodeMessage,idNodeStart+LEN(ID_NODE_PREFIX)-1,1);
posSeparator:=FINDP(partialStringNode, FIELD_SEPARATOR,1);
idNode:=STRING_TO_WORD(MID(partialStringNode,posSeparator-1,1));

(*get node id - PW0*)
idPw0Start:=FINDP(statusNodeMessage,PW0_PREFIX,1);
partialStringPW0:=DELETE(statusNodeMessage,idPw0Start+LEN(PW0_PREFIX)-1,1);
posSeparator:=FINDP(partialStringPW0, FIELD_SEPARATOR,1);
pwm0:=STRING_TO_WORD(MID(partialStringPW0,posSeparator-1,1));

(*get node id - PW1*)
idPw1Start:=FINDP(statusNodeMessage,PW1_PREFIX,1);
partialStringPW1:=DELETE(statusNodeMessage,idPw1Start+LEN(PW1_PREFIX)-1,1);
posSeparator:=FINDP(partialStringPW1, FIELD_SEPARATOR,1);
pwm1:=STRING_TO_WORD(MID(partialStringPW1,posSeparator-1,1));

(*get node id - PW2*)
idPw2Start:=FINDP(statusNodeMessage,PW2_PREFIX,1);
partialStringPW2:=DELETE(statusNodeMessage,idPw2Start+LEN(PW2_PREFIX)-1,1);
posSeparator:=FINDP(partialStringPW2, FIELD_SEPARATOR,1);
pwm2:=STRING_TO_WORD(MID(partialStringPW2,posSeparator-1,1));

state.id_Geolumen:=idNode;
state.DimmValue_0:=pwm0;
state.DimmValue_1:=pwm1;
state.DimmValue_2:=pwm2;
END_ACTION
ACTION ReadID:
(* Ricerca tra i messaggi arrivati quali sono settati come DATAREC e quindi usa i dati per definire l'ID associato a quel lux e depositarlo nella struttura TabListLux *)
FOR counter:= 0 TO MAX_ARRAY_MSG DO
	IF ( MsgRecBuffer[counter].MsgType = DATAREC AND   FIND(MsgRecBuffer[counter].Msg,  'NMEAS;MAC' ) = 4 ) AND ( FIND(MsgRecBuffer[counter].Msg,  'IDN' ) = 30) THEN
		StrSaveMacAdd:=MID(MsgRecBuffer[counter].Msg, 8 , 21);
		StrLoc:=33;
		Str := MID(MsgRecBuffer[counter].Msg, 1 , StrLoc);
		WHILE Str <> ';' DO (*Cerco il numero IDN e lo memorizzo in StrSaveID dopo il while*)
			StrLoc:=StrLoc+1;
			Str := MID(MsgRecBuffer[counter].Msg, 1 , StrLoc);
		END_WHILE
		StrSaveID:=MID(MsgRecBuffer[counter].Msg, StrLoc-33 , 33);
		index:=1;
		WHILE (index<=MAX_LUXNUM) AND (SysStrCmp(TabListLux[index].StMacAdd,  StrSaveMacAdd) <> 0)   DO (*diego setting *)
			index:= index +1;
		END_WHILE
		IF index<=MAX_LUXNUM THEN
			TabListLux[index].xCoupled := TRUE; (*Indico che ho accoppiato l'ID con il mac address*)
			TabListLux[index].LuxID_Geolumen:=STRING_TO_WORD(StrSaveID); (*Salvo l'ID accoppiato al mac address - info che sarà poi da spedire al server*)
			LuxElement[index].ID := TabListLux[index].LuxNumber; (*  copio id del lux nella tabella delle variabili dei lux *)
			IF LuxElement[index].CTRL_MODE = 2 THEN
				(* init astro *)
				ASTR[index](ID:= LuxElement[index].ID, localTime:=Sys.Time_CT_DT);
				ASTR_CONFIG[index].ID:=ASTR[index].ID;
			END_IF
			LuxGeolumenNodes[index].ID_Geolumen:=TabListLux[index].LuxID_Geolumen;
			LuxGeolumenNodes[index].ID_Lux:=LuxElement[index].ID ;
		END_IF
	END_IF
END_FOR
END_ACTION
ACTION SendAuth:
FOR i:=0 TO ArrayPos DO
	IF MsgRecBuffer[i].MsgType = REQAUTH0 THEN
		MacStr:=MID(MsgRecBuffer[i].Msg, 8, 23); (*Isolo la sottostringa del Mac address - es. 0046CD12*)

		FOR x:= 1 TO MAX_LUXNUM DO
			IF SysStrCmp(MacStr, TabListLux[x].StMacAdd) = 0 THEN
				 (*spedisci autorizzazione   CMD_ADD_NODE:21:36096:70:50744$0D$0A  *)
				StrToSend:=CONCAT('CMD_ADD_NODE:21:36096:', WORD_TO_STRING(TabListLux[x].MacAddH) );
				StrToSend:=CONCAT(StrToSend, ':');
				StrToSend:=CONCAT(StrToSend,  WORD_TO_STRING(TabListLux[x].MacAddL) );
				StrToSend:=CONCAT(StrToSend,  '$R$N' );
				(*SendData(pTxData:=ADR(StrToSend));*)
				SendDataQueue(pTxData:=ADR(StrToSend));
				SendDataQueue.addMessage();
				SendDataQueue();
				MsgRecBuffer[i].MsgType:=COMPLETED;
				x:=  MAX_LUXNUM+1;
			END_IF
		END_FOR
	END_IF
END_FOR
END_ACTION
ACTION testFakeReadID:
(* Ricerca tra i messaggi arrivati quali sono settati come DATAREC e quindi usa i dati per definire l'ID associato a quel lux e depositarlo nella struttura TabListLux *)
FOR counter:= 0 TO MAX_ARRAY_MSG DO
	IF ( MsgRecBuffer[counter].MsgType = DATAREC AND   FIND(MsgRecBuffer[counter].Msg,  'NMEAS;MAC' ) = 4 ) AND ( FIND(MsgRecBuffer[counter].Msg,  'IDN' ) = 30) THEN
		StrSaveMacAdd:=MID(MsgRecBuffer[counter].Msg, 8 , 21);
		StrLoc:=33;
		Str := MID(MsgRecBuffer[counter].Msg, 1 , StrLoc);
		WHILE Str <> ';' DO (*Cerco il numero IDN e lo memorizzo in StrSaveID dopo il while*)
			StrLoc:=StrLoc+1;
			Str := MID(MsgRecBuffer[counter].Msg, 1 , StrLoc);
		END_WHILE
		StrSaveID:=MID(MsgRecBuffer[counter].Msg, StrLoc-33 , 33);
		index:=1;
		WHILE (index<=MAX_LUXNUM) AND (SysStrCmp(TabListLux[index].StMacAdd,  StrSaveMacAdd) <> 0)   DO (*diego setting *)
			index:= index +1;
		END_WHILE
		IF index<=MAX_LUXNUM THEN
			TabListLux[index].xCoupled := TRUE; (*Indico che ho accoppiato l'ID con il mac address*)
			TabListLux[index].LuxID_Geolumen:=STRING_TO_WORD(StrSaveID); (*Salvo l'ID accoppiato al mac address - info che sarà poi da spedire al server*)
			LuxElement[index].ID := TabListLux[index].LuxNumber; (*  copio id del lux nella tabella delle variabili dei lux *)
			IF LuxElement[index].CTRL_MODE = 2 THEN
				(* init astro *)
				ASTR[index](ID:= LuxElement[index].ID, localTime:=Sys.Time_CT_DT);
				ASTR_CONFIG[index].ID:=ASTR[index].ID;
			END_IF
			LuxGeolumenNodes[index].ID_Geolumen:=TabListLux[index].LuxID_Geolumen;
			LuxGeolumenNodes[index].ID_Lux:=LuxElement[index].ID ;
		END_IF
	END_IF
END_FOR
END_ACTION
ACTION updateNetworkTime:
			StrMin:=BYTE_TO_STRING(Sys.Time_Min);
			IF  Sys.Time_Min<=9 THEN
				StrMin := CONCAT('0',StrMin);
			END_IF
			StrMin:=MID(STR:=StrMin, LEN:=2, POS:= 1);
			StrHour:=BYTE_TO_STRING(Sys.Time_Hour);
			IF Sys.Time_Hour<=9 THEN
				StrHour := CONCAT('0',StrHour);
			END_IF
			StrHour:=MID(STR:=StrHour, LEN:=2, POS:= 1);

			(* aggiorno l'ora del coordinatore e della rete *)
			SendString := 'NWK_TIME_SET=$R$N';
			SendString :=INSERT (SendString,StrHour,13);
			SendString :=INSERT (SendString,':',15);
			SendString :=INSERT (SendString,StrMin,16);
			xStartSend := TRUE;

			SendDataQueue(pTxData:=ADR(SendString),ReceiveBufferPtr:=ADR(ReceiveBuffer));
			SendDataQueue.addMessage();
			SendDataQueue();
END_ACTION

(* POU GeoLumenWrapping/getGeolumenNodeByGeolumenId, ST *)
FUNCTION getGeolumenNodeByGeolumenId : INT
VAR_INPUT
	GeolumenId : INT;
END_VAR

VAR
	I : INT;
END_VAR
getGeolumenNodeByGeolumenId:=-1;
FOR I:=1 TO MAX_LUXNUM DO
	IF (LuxGeolumenNodes[i].ID_Geolumen = GeolumenId) THEN getGeolumenNodeByGeolumenId :=i; RETURN; END_IF
END_FOR
END_FUNCTION

(* POU GeoLumenWrapping/SendData, ST *)
FUNCTION SendData : BOOL
VAR_INPUT
	pTxData: POINTER TO STRING;
END_VAR
VAR

	StrToSend		: STRING;
	xOpenPort		: BOOL := TRUE;
	xInitPort			: BOOL;
	xStartSend		: BOOL;
	xSendActive	: BOOL;

	pRecStr 	: POINTER TO STRING(255);
	StringFromCom 	: STRING(255);
	tmpStringa : STRING(255) := '';
	LastMsg: STRING(255) := '';

	intStart, x : INT;
	counterFrame : INT :=0;
END_VAR
StrToSend:=pTxData^;
xSendActive:= TRUE;
COM0(	utRECEIVE_BUFFER := ReceiveBuffer,
		ptSEND_BUFFER	:= ADR(StrToSend),
		xINIT				:=  xInitPort,
     		xOPEN_COM_PORT 	:= xOpenPort,
		iBYTES_TO_SEND	:= LEN(StrToSend)+1,
		xSTART_SEND		:= xSendActive );
END_FUNCTION

(* POU GeoLumenWrapping/isGeolumenIEqualStatus, ST *)
FUNCTION isGeolumenIEqualStatus : BOOL
VAR_INPUT
	desideredState: type_LuxGeolumenStatus;
	feedbackState: type_LuxGeolumenStatus;
END_VAR
VAR
END_VAR
isGeolumenIEqualStatus:=(desideredState.ID_Geolumen=feedbackState.ID_Geolumen) AND
					  (desideredState.DimmValue_0=feedbackState.DimmValue_0) AND
 					  (desideredState.DimmValue_1=feedbackState.DimmValue_1) AND
					  (desideredState.DimmValue_2=feedbackState.DimmValue_2) ;
END_FUNCTION

(* POU PLANT_PROCESS/SCA_Proc, ST *)
PROGRAM SCA_Proc
VAR

	fCoord		:FLT_TAP;  (* geolumen coord STATUS *)
	(*SCA01_1	:	FLT_TAP;
	SCA01_2	:	FLT_TAP;
	SCA01_3	:	FLT_TAP;

	upd		:	BOOL;*)
END_VAR
(*### geolumen COORD Status Check ###*)
fCoord(IN:=COORD_STATUS);
IF fCoord.EVH THEN
	LogEv(EL_Log,EO_VPN,1,3,'GEOLUMEN_COORD_STATUS_UP');
END_IF
IF fCoord.EVL THEN
	LogEv(EL_Wrn,EO_VPN,1,4,'GEOLUMEN_COORD_STATUS_DOWN');
END_IF
(***** SCA01 *****)
(*SCA01_1(IN:=SCA01_1_DI);
IF SCA01_1.EVL THEN LogEv(EL_Wrn,EO_SCA,1,1,'1'); upd:=TRUE; END_IF
IF SCA01_1.EVH THEN	LogEv(EL_Log,EO_SCA,1,2,'1'); upd:=TRUE; END_IF

SCA01_2(IN:=SCA01_2_DI);
IF SCA01_2.EVL THEN	LogEv(EL_Wrn,EO_SCA,1,1,'2'); upd:=TRUE; END_IF
IF SCA01_2.EVH THEN	LogEv(EL_Log,EO_SCA,1,2,'2'); upd:=TRUE; END_IF

SCA01_3(IN:=SCA01_3_DI);
IF SCA01_3.EVL THEN	LogEv(EL_Wrn,EO_SCA,1,1,'3'); upd:=TRUE; END_IF
IF SCA01_3.EVH THEN	LogEv(EL_Log,EO_SCA,1,2,'3'); upd:=TRUE; END_IF

IF upd THEN
	upd:=FALSE;
	Logger_Head();
	AddLogData();
	Logger_Send();
END_IF*)
;
END_PROGRAM
ACTION AddLogData:
(*Logger.s1:='&SCA01=';
Logger.s1:=CONCAT(Logger.s1,BYTE_TO_STRING(BOOL_TO_BYTE(SCA01_1.OUT))		); Logger.s1:=CONCAT(Logger.s1,';');
Logger.s1:=CONCAT(Logger.s1,BYTE_TO_STRING(BOOL_TO_BYTE(SCA01_2.OUT))		); Logger.s1:=CONCAT(Logger.s1,';');
Logger.s1:=CONCAT(Logger.s1,BYTE_TO_STRING(BOOL_TO_BYTE(SCA01_3.OUT))		);
ADDSTRING(ADR(Logger.TData), ADR(Logger.s1), Logger.TLen);*)
;
END_ACTION

(* POU PLANT_PROCESS/SYS_Proc, ST *)
PROGRAM SYS_Proc
VAR
	fVPN_ST2		:FLT_TAP;  (* VPN STATUS *)
(*	fKEY_CT_ST		:FLT_TAP; (* DOOR01 - Porta primaria *)*)
(*	fKEY_SCT_ST		:FLT_TAP; (* DOOR02 - Porta secondaria *)*)

END_VAR
(*### VPN Status Check ###*)
fVPN_ST2(IN:=VPN_STATUS);
IF fVPN_ST2.EVH THEN
	LogEv(EL_Log,EO_VPN,1,3,'STATUS_UP');
END_IF
IF fVPN_ST2.EVL THEN
	LogEv(EL_Wrn,EO_VPN,1,4,'STATUS_DOWN');
END_IF
END_PROGRAM

(* POU PLANTCONFIG/addAllAstroLog, ST *)
FUNCTION addAllAstroLog : BOOL
VAR_INPUT
	astroLength :WORD;
END_VAR
VAR
	groupSize: WORD:=10; (*FACTOR OF GROUPING*)
	groupNumber : WORD;
	i : WORD;
	j : WORD;
	index:WORD;
	isObj : BOOL;
END_VAR
groupNumber:=astroLength/groupSize;
IF((astroLength MOD groupSize) <>0) THEN groupNumber:=groupNumber+1; END_IF

FOR i:=0 TO groupNumber-1 DO
	(*verifico se nel gruppo corrente c'è qualche ASTR valido *)
	isObj:=FALSE;
	FOR j:=0 TO groupSize-1 DO
		index:=i*groupNumber+j;
		IF(index<>0 AND index<=astroLength AND ASTR[index].ID<>0 ) THEN isObj:=TRUE; j:=groupSize; END_IF
	END_FOR
	(* se c'è qualche ASTR valido da fare, procedo *)
	IF(isObj) THEN
		Logger_Head();
		FOR j:=0 TO groupSize-1 DO
			index:=i*groupNumber+j;
			IF(index<>0 AND index<=astroLength AND ASTR[index].ID<>0 ) THEN ASTR[index].AddLogData(); END_IF
		END_FOR
		IF(i=groupNumber-1 AND (index+1)<=astroLength AND ASTR[index+1].ID<>0)  THEN ASTR[index+1].AddLogData(); END_IF
		Logger_Send();
	END_IF
END_FOR
END_FUNCTION

(* POU PLANTCONFIG/addAllLuxLog, ST *)
FUNCTION addAllLuxLog : BOOL
VAR_INPUT
	luxLength : WORD;
END_VAR
VAR
	groupSize: WORD:=10; (*FACTOR OF GROUPING*)
	groupNumber : WORD;
	i : WORD;
	j : WORD;
	index:WORD;
	isObj : BOOL;
END_VAR
groupNumber:=luxLength/groupSize;
IF((luxLength MOD groupSize) <>0) THEN groupNumber:=groupNumber+1; END_IF

FOR i:=0 TO groupNumber-1 DO
	(*verifico se nel gruppo corrente c'è qualche ASTR valido *)
	isObj:=FALSE;
	FOR j:=0 TO groupSize-1 DO
		index:=i*groupNumber+j;
		IF(index<>0 AND index<=luxLength AND LuxElement[index].ID<>0 ) THEN isObj:=TRUE; j:=groupSize; END_IF
	END_FOR
	(* se c'è qualche ASTR valido da fare, procedo *)
	IF(isObj) THEN
		Logger_Head();
		FOR j:=0 TO groupSize-1 DO
			index:=i*groupNumber+j;
			IF(index<>0 AND index<=luxLength AND LuxElement[index].ID<>0 ) THEN

				LuxElement[index].AddLogData(WORKINGTIME:=GlobalWorkingtime	[index],
									    POWERONCYCLES:=GlobalPowerOnCycles[index],
									    ENERGYCOUNTER:=GlobalEnergyCounter[index],
									    ENERGYCOUNTER_t :=GlobalEnergyCounter_t[index]);
			END_IF
		END_FOR
		IF(i=groupNumber-1 AND (index+1)<=luxLength AND LuxElement[index+1].ID<>0)  THEN

				LuxElement[index].AddLogData(WORKINGTIME:=GlobalWorkingtime	[index],
									    POWERONCYCLES:=GlobalPowerOnCycles[index],
									    ENERGYCOUNTER:=GlobalEnergyCounter[index],
									    ENERGYCOUNTER_t :=GlobalEnergyCounter_t[index]);
		END_IF
		Logger_Send();
	END_IF
END_FOR
END_FUNCTION

(* POU GeoLumenWrapping/GeolumenNodeList, ST *)
FUNCTION_BLOCK GeolumenNodeList (*Esegue la lettura dei mac address e del numero id associato nel file x_Lux_List.txt dove x è il numero id del plc*)
VAR_OUTPUT
	Message		: STRING;
END_VAR
VAR CONSTANT
	RTS_INVALID_HANDLE : DWORD:=0;
	AM_READ: STRING [20]:= 'r';			(* Use 'w' (write), 'r' (read) or 'rw' (read and write) *)
	MAX_LINE_CHARLEN:WORD:=100;
END_VAR
VAR
	(*hMode		: ACCESS_MODE;
	hFile		: RTS_IEC_HANDLE;
	hRes		: RTS_IEC_RESULT;  *)
	bList		: ARRAY [0..MAX_LINE_CHARLEN] OF BYTE;
	bListLen :INT;
	hFile		: DWORD;

	i, j			: DWORD;
	k, x			: INT;
	xwDimFile	: LWORD;
	bChar		: BYTE;
	sFileName 	: STRING;
	ValueToInsert: WORD;
	wLocal		: WORD;
	bIndex:INT;
	lastPosSeparator:INT;
	pot:WORD;
	xRel:INT;
END_VAR
Message:='';
bIndex:=0;
lastPosSeparator:=0;
pot:=0;
FOR i:=0 TO MAX_LINE_CHARLEN DO
	BList[i]:=0;
END_FOR
hfile:=0;
(* Open data file *)
sFileName:=CONCAT(STR1:=MapConf_Path, STR2:=PLC_ID);
sFileName:=CONCAT(STR1:=sFileName, STR2:=Luxlist_FileName);
hFile:=SysFileOpen(sFileName,AM_READ);

(* File not found *)
IF hFile=RTS_INVALID_HANDLE THEN
	Message:='File not found';
	RETURN;
END_IF

(* Close file *)
SysFileClose(hFile);

(* Open data file *)
i:=0;
j:=0;
k:=0;
x:=0;
bListLen:=0;
wLocal:=0;
ValueToInsert:=0;
bChar:=0;
xwDimFile:=0;
hFile:=SysFileOpen(sFileName,AM_READ);

SysFileSetPos(hFile, i);
SysFileRead(hFile, ADR(bList[j]), 1);

(* WHILE NOT (SysFileEOF(hFile)) DO  *)
REPEAT
	IF bList[j] = 16#2F  (* se trovo '/'  *)
		THEN
			SysFileSetPos(hFile, i+1);
			SysFileRead(hFile, ADR(bList[j+1]), 1);
			IF bList[j+1] = 16#2F (* se trovo ancora '/'  *)
				THEN
					WHILE  bList[j]<> 16#0D DO
						i := i+1;
						SysFileSetPos(hFile, i);	
						SysFileRead(hFile, ADR(bList[j]), 1);
					END_WHILE
					i := i+1;
					SysFileSetPos(hFile, i);
					SysFileRead(hFile, ADR(bList[j]), 1);
					IF bList[j] = 16#0A
						THEN 
							i := i+1;
							j := 0;
							SysFileSetPos(hFile, i);	
							SysFileRead(hFile, ADR(bList[j]), 1); (*leggo il primo carattere della nuova riga  *)
						ELSE
							Message:='Errore 0D 0A';
							RETURN;
					END_IF
				ELSE
					Message:='Errore //';
					RETURN;
			END_IF
	END_IF
	IF bList[j] <> 16#3B (*finchè non trovo ;   *)
		THEN
			IF bList[j] = 16#2C THEN
				lastPosSeparator:=DWORD_TO_INT(j);
			END_IF
			i:=i+1;
			j:=j+1;
			bListLen:=bListLen+1;
		ELSE
			i:=i+3;   (* Se trovo ; inizio a salvare i dati della riga letta in TabListLux[k]....  *)
			j:=0;
			k:=k+1;
			FOR bIndex:=0 TO lastPosSeparator-1 DO
				pot:=lastPosSeparator-1 -bIndex;
				TabListLux[k].LuxNumber :=TabListLux[k].LuxNumber+BYTE_TO_DWORD(bList[bIndex]-16#30)*REAL_TO_DWORD(EXPT(10,pot)) ;  (*   memorizzo il numero del lux   *)
			END_FOR
			TabListLux[k].StMacAdd:='';
			FOR x:=lastPosSeparator+1 TO bListLen-1 DO
				CASE bList[x] OF
					16#61: bList[x]:=16#41;
					16#62: bList[x]:=16#42;
					16#63: bList[x]:=16#43;
					16#64: bList[x]:=16#44;
					16#65: bList[x]:=16#45;
					16#66: bList[x]:=16#46;
				END_CASE
				TabListLux[k].StMacAdd:= CONCAT(TabListLux[k].StMacAdd, ASCIIBYTE_TO_STRING(bList[x]));
			END_FOR
			FOR x:=lastPosSeparator+1 TO lastPosSeparator+1+3  DO
				xRel:=x-(lastPosSeparator+1);
				 IF( bList[x]<=16#39 AND  bList[x]>=16#30)
				THEN
					wLocal:=BYTE_TO_WORD(bList[x]-16#30);
					TabListLux[k].MacAddH :=  TabListLux[k].MacAddH + SHL(wLocal, 12-(xRel)*4); (* Corrisponde a  4*(7-x)   *)
				ELSE

					CASE  bList[x] OF
						16#61, 16#41:
							ValueToInsert:= 16#0A;
							TabListLux[k].MacAddH :=  TabListLux[k].MacAddH + SHL( ValueToInsert, 12-(xRel)*4);
						16#62, 16#42:
							ValueToInsert:= 16#0B;
							TabListLux[k].MacAddH :=  TabListLux[k].MacAddH + SHL( ValueToInsert, 12-(xRel)*4);
						16#63, 16#43:
							ValueToInsert:= 16#0C;
							TabListLux[k].MacAddH :=  TabListLux[k].MacAddH + SHL( ValueToInsert, 12-(xRel)*4);
						16#64, 16#44:
							ValueToInsert:= 16#0D;
							TabListLux[k].MacAddH :=  TabListLux[k].MacAddH + SHL( ValueToInsert, 12-(xRel)*4);
						16#65, 16#45:
							ValueToInsert:= 16#0E;
							TabListLux[k].MacAddH :=  TabListLux[k].MacAddH + SHL( ValueToInsert, 12-(xRel)*4);
						16#66, 16#46:
							ValueToInsert:= 16#0F;
							TabListLux[k].MacAddH :=  TabListLux[k].MacAddH + SHL( ValueToInsert, 12-(xRel)*4);
					END_CASE
				END_IF
			END_FOR
			FOR x:=lastPosSeparator+1+4 TO lastPosSeparator+1+4+3 DO
				xRel:=x-(lastPosSeparator+1+4);
				 IF( bList[x]<=16#39 AND  bList[x]>=16#30)
				THEN
					wLocal:=BYTE_TO_WORD(bList[x]-16#30);
					TabListLux[k].MacAddL :=  TabListLux[k].MacAddL + SHL(wLocal, 12-(xRel)*4); (* Corrisponde a  4*(7-x)   *)
				ELSE

					CASE  bList[x] OF
						16#61, 16#41:
							ValueToInsert:= 16#0A;
							TabListLux[k].MacAddL :=  TabListLux[k].MacAddL + SHL( ValueToInsert, 12-(xRel)*4);
						16#62, 16#42:
							ValueToInsert:= 16#0B;
							TabListLux[k].MacAddL :=  TabListLux[k].MacAddL + SHL( ValueToInsert, 12-(xRel)*4);
						16#63, 16#43:
							ValueToInsert:= 16#0C;
							TabListLux[k].MacAddL :=  TabListLux[k].MacAddL + SHL( ValueToInsert, 12-(xRel)*4);
						16#64, 16#44:
							ValueToInsert:= 16#0D;
							TabListLux[k].MacAddL :=  TabListLux[k].MacAddL + SHL( ValueToInsert, 12-(xRel)*4);
						16#65, 16#45:
							ValueToInsert:= 16#0E;
							TabListLux[k].MacAddL :=  TabListLux[k].MacAddL + SHL( ValueToInsert, 12-(xRel)*4);
						16#66, 16#46:
							ValueToInsert:= 16#0F;
							TabListLux[k].MacAddL :=  TabListLux[k].MacAddL + SHL( ValueToInsert, 12-(xRel)*4);
					END_CASE
				END_IF
			END_FOR
			TabListLux[k].MacAdd:=SHL(TabListLux[k].MacAddH, 16)+TabListLux[k].MacAddL;
			bListLen:=0;
			lastPosSeparator:=0;
			pot:=0;
	END_IF
	SysFileSetPos(hFile, i);
	SysFileRead(hFile, ADR(bList[j]), 1);
UNTIL  ((SysFileEOF(hFile)) AND ( bList[j] <> 16#3B))
END_REPEAT
(* END_WHILE  *)
IF SysFileEOF(hFile) = 0
	THEN Message:='Reading Default_Lux File: OK';
END_IF

(* Close file *)
SysFileClose(hFile);
END_FUNCTION_BLOCK

(* POU GeoLumenWrapping/GeolumenSaveTabListLux, ST *)
FUNCTION GeolumenSaveTabListLux  : BOOL
VAR
	hName : STRING(255) :='TABLISTLUX.TXT';
	hFile	 : DWORD;
	i	 : INT;
	line:STRING(255):='';
	tmp:STRING(8):='';
	macString:STRING(8);
	count:INT:=0;
	refCount:INT:=0;
END_VAR
count:=0;
FOR i := 1 TO MAX_LUXNUM  DO
	IF  LuxElement[i].ID <> 0  THEN
		count:=count+1;
	END_IF
END_FOR
refCount:=count;
count:=0;
hName:=CONCAT(FilesPath ,hName);
hFile:=SysFileOpen(hName,'w');
IF hFile<>0 THEN
	FOR i := 1 TO MAX_LUXNUM  DO
		IF  LuxElement[i].ID <> 0  THEN
			count:=count+1;
			line:=CONCAT(DWORD_TO_STRING(TabListLux[i].LuxNumber),',');
			tmp:=DWORD_TO_STRH(TabListLux[i].MacAdd);
			line:=CONCAT(line,tmp);
			line:=CONCAT(line,';');
			IF count < refCount THEN line:=CONCAT(line,'$R$N'); END_IF
			SysFileWrite(hFile, ADR(line),LEN(line));
		END_IF
	END_FOR
	SysFileClose(hFile);
END_IF
END_FUNCTION

(* POU GeoLumenWrapping/getGeolumenIDbyLuxID, ST *)
FUNCTION getGeolumenIDbyLuxID : DWORD
VAR_INPUT
	LuxID:WORD;
END_VAR
VAR
	i:INT;
END_VAR
IF LuxID = 0 THEN
	getGeolumenIDbyLuxID:=0;
END_IF
FOR i:=1 TO MAX_LUXNUM DO
	IF TabListLux[i].LuxNumber=LuxID THEN
		getGeolumenIDbyLuxID:=TabListLux[i].LuxID_Geolumen;
		RETURN;
	END_IF
END_FOR
END_FUNCTION

(* POU GeoLumenWrapping/getGeolumenNodeByLuxId, ST *)
FUNCTION getGeolumenNodeByLuxId : INT
VAR_INPUT
	LuxID : INT;
END_VAR

VAR
	I : INT;
END_VAR
getGeolumenNodeByLuxId:=-1;
FOR I:=1 TO MAX_LUXNUM DO
	IF (LuxGeolumenNodes[i].ID_Lux = LuxID) THEN getGeolumenNodeByLuxId :=i; RETURN; END_IF
END_FOR
END_FUNCTION

(* POU GeoLumenWrapping/getLuxIDbyGeolumenID, ST *)
FUNCTION getLuxIDbyGeolumenID : DWORD
VAR_INPUT
	GeolumenID:WORD;
END_VAR
VAR
	i:INT;
END_VAR
IF GeolumenID = 0 THEN
	getLuxIDbyGeolumenID:=0;
END_IF
FOR i:=1 TO MAX_LUXNUM DO
	IF TabListLux[i].LuxID_Geolumen=GeolumenID THEN
		getLuxIDbyGeolumenID:=TabListLux[i].LuxNumber;
		RETURN;
	END_IF
END_FOR
END_FUNCTION

(* POU PLANTCONFIG/isValidLuxID, ST *)
FUNCTION isValidLuxID : BOOL
VAR_INPUT
	id: WORD;
END_VAR
VAR
END_VAR
isValidLuxID:=id>=1 AND id<=MAX_LUXNUM;
IF(isValidLuxID) THEN isValidLuxID:=(LuxElement[id].ID <> 0); END_IF
END_FUNCTION

(* POU GeoLumenWrapping/LuxGeolumenDiagnostics, ST *)
FUNCTION_BLOCK LuxGeolumenDiagnostics
VAR_INPUT
	turnOnRequest:BOOL;
	turnOffRequest:BOOL;
	restoreAllRequest:BOOL;
	executeCommandRequest:BOOL;
	executeCommandSetRequest:BOOL;
	executeCommandGetRequest:BOOL;
	executeCommandGetIDByMACRequest:BOOL;
	executeCommandGetMACByIDRequest:BOOL;
	executeCommandResetRequest:BOOL;
	executeCommandSaveToFileRequest:BOOL;
	commandSetID:WORD;
	commandGetID:STRING(10):='';
	commandSetDIMM:INT;
	commandGetIDByMac:DWORD;
	commandGetIDByMacResult:DWORD;
	commandGetMacByID:WORD	;
	commandGetMacByIDResult:DWORD;
	diagnosticCommand:STRING(255):='';
END_VAR
VAR
	LuxCount:WORD;
	COUNT:INT:=0;
	I:INT:=0;
END_VAR
IF restoreAllRequest THEN
	restoreAll();
	restoreAllRequest:=FALSE;
END_IF
IF turnOnRequest THEN
	turnOnAll();
	turnOnRequest:=FALSE;
END_IF
IF turnOffRequest THEN
	turnOffAll();
	turnOffRequest:=FALSE;
END_IF
IF executeCommandRequest THEN
	executeCommand();
	executeCommandRequest:=FALSE;
END_IF
IF executeCommandSetRequest THEN
	executeSetCommand();
	executeCommandSetRequest:=FALSE;
END_IF
IF executeCommandGetRequest THEN
	executeGetCommand();
	executeCommandGetRequest:=FALSE;
END_IF
IF executeCommandGetIDByMACRequest THEN
	executeGetCommandIDByMAC();
	executeCommandGetIDByMACRequest:=FALSE;
END_IF
IF executeCommandGetMACByIDRequest THEN
	executeGetCommandMACByID();
	executeCommandGetMACByIDRequest:=FALSE;
END_IF
IF executeCommandResetRequest THEN
	executeCommandReset();
	executeCommandResetRequest :=FALSE;
END_IF
IF executeCommandSaveToFileRequest THEN
	GeolumenSaveTabListLux();
	executeCommandResetRequest :=FALSE;
END_IF
END_FUNCTION_BLOCK
ACTION executeCommand:
IF FIND(diagnosticCommand,'$R$N') <1 THEN diagnosticCommand:=CONCAT(diagnosticCommand,'$R$N'); END_IF
SendDataQueue(pTxData:=ADR(diagnosticCommand),ReceiveBufferPtr:=ADR(ReceiveBuffer));
SendDataQueue.addMessage();
SendDataQueue();
END_ACTION
ACTION executeCommandReset:
diagnosticCommand:='CMD_SW_RESET$R$N';
SendDataQueue(pTxData:=ADR(diagnosticCommand),ReceiveBufferPtr:=ADR(ReceiveBuffer));
SendDataQueue.addMessage();
SendDataQueue();
diagnosticCommand:='CMD_AUTHORISE=0$R$N';
SendDataQueue(pTxData:=ADR(diagnosticCommand),ReceiveBufferPtr:=ADR(ReceiveBuffer));
SendDataQueue.addMessage();
SendDataQueue();
END_ACTION
ACTION executeGetCommand:
diagnosticCommand:='NDE_GET_STATUS=x$R$N';
diagnosticCommand:=REPLACE_ALL(diagnosticCommand,'x',commandGetID);

SendDataQueue(pTxData:=ADR(diagnosticCommand),ReceiveBufferPtr:=ADR(ReceiveBuffer));
SendDataQueue.addMessage();
SendDataQueue();
END_ACTION
ACTION executeGetCommandIDByMAC:
FOR LuxCount:=1 TO  MAX_LUXNUM DO
	IF  TabListLux[LuxCount].MacAdd<>0 AND TabListLux[LuxCount].MacAdd=commandGetIDByMac THEN
			commandGetIDByMacResult:=TabListLux[LuxCount].LuxNumber;
			RETURN;
	END_IF
END_FOR
END_ACTION
ACTION executeGetCommandMACByID:
FOR LuxCount:=1 TO  MAX_LUXNUM DO
	IF  TabListLux[LuxCount].LuxNumber<>0 AND TabListLux[LuxCount].LuxNumber=commandGetMacByID THEN
		commandGetMacByIDResult:=TabListLux[LuxCount].MacAdd;
		RETURN;
	END_IF
END_FOR
END_ACTION
ACTION executeSetCommand:
FOR i:=1 TO MAX_LUXNUM DO
		IF LuxElement[i].ID=commandSetID THEN

			IF(commandSetDIMM>0) THEN
					LuxElement [i] . CTRL_MODE := 1 ; (*// Set to manuale on con dimm*)
					LuxElement [i].DimmingValForManual:=commandSetDIMM;
			ELSE
					LuxElement [i] . CTRL_MODE := 0 ; (*// Set to manuale off*)
					LuxElement [i].DimmingValForManual:=0;
			END_IF

			LuxElement [  i  ] (     WORKINGTIME := GlobalWorkingTime [ i ] ,
			POWERONCYCLES:= GlobalPowerOnCycles [  i  ] ,
			ENERGYCOUNTER :=GlobalEnergyCounter [  i ] ,
			ENERGYCOUNTER_T :=GlobalEnergyCounter_t [  i  ] ,
									CtrlExton := KEYON ) ;
		END_IF
END_FOR
END_ACTION
ACTION restoreAll:
FOR LuxCount:=1 TO  MAX_LUXNUM DO
	IF  LuxElement[LuxCount].ID <> 0  THEN

		LuxElement [  LuxCount ] . CTRL_MODE := LuxElement [ LuxCount] . CTRL_MODE_backUp ;
		LuxElement [  LuxCount ] (     WORKINGTIME := GlobalWorkingTime [ LuxCount ] ,
							POWERONCYCLES :=
							GlobalPowerOnCycles [ LuxCount ] ,
							ENERGYCOUNTER := GlobalEnergyCounter [ LuxCount ] ,
							ENERGYCOUNTER_T :=
							GlobalEnergyCounter_t [ LuxCount ] ,
							CtrlExton := KEYON ) ;
	END_IF
END_FOR
END_ACTION
ACTION turnOffAll:
FOR LuxCount:=1 TO  MAX_LUXNUM DO
	IF  LuxElement[LuxCount].ID <> 0  THEN

					LuxElement [ LuxCount ] . CTRL_MODE := 0 ; (*// Set to manuale OFF *)
					LuxElement [ LuxCount ].DimmingValForManual:=0;
					LuxElement [ LuxCount ] (     WORKINGTIME := GlobalWorkingTime [ LuxCount ] ,
									POWERONCYCLES:= GlobalPowerOnCycles [ LuxCount ] ,
									ENERGYCOUNTER :=GlobalEnergyCounter [ LuxCount ] ,
									ENERGYCOUNTER_T :=GlobalEnergyCounter_t [ LuxCount ] ,
									CtrlExton := KEYON ) ;
	END_IF
END_FOR
END_ACTION
ACTION turnOnAll:
FOR LuxCount:=1 TO  MAX_LUXNUM DO
	IF  LuxElement[LuxCount].ID <> 0  THEN

					LuxElement [ LuxCount  ] . CTRL_MODE := 1 ; (*// Set to manuale ON *)
					LuxElement [ LuxCount ].DimmingValForManual:=LuxElement [ LuxCount ].MAX_DIMM_VALUE;
					LuxElement [ LuxCount] (     WORKINGTIME := GlobalWorkingTime [ LuxCount ] ,
									POWERONCYCLES:= GlobalPowerOnCycles [ LuxCount ] ,
									ENERGYCOUNTER :=GlobalEnergyCounter [ LuxCount ] ,
									ENERGYCOUNTER_T :=GlobalEnergyCounter_t [ LuxCount ] ,
									CtrlExton := KEYON ) ;
	END_IF
END_FOR
END_ACTION

(* POU GeoLumenWrapping/obj_GeolumenNode, ST *)
FUNCTION_BLOCK obj_GeolumenNode
VAR CONSTANT
	MAX_NO_FEEDBACK_TIME:TIME:=t#3m; (*minutes*)
	MAX_RETRY_NO_FEEDBACK:BYTE:=5;
	MAX_RETRY_STATUS_NOT_ALIGNED:BYTE:=10;
END_VAR

VAR_INPUT
	ID_Geolumen: DWORD;
	ID_LUX: DWORD;
	desideredDimmValue:WORD;
	feedbackState: type_LuxGeolumenStatus;
	lastSeen:DT;
END_VAR
VAR CONSTANT
	MIN_DIMM:WORD:=0;
	MAX_DIMM:WORD:=1023;
	MAX_DIMM_LUX_CLEVERGY:WORD:=100;
END_VAR
VAR_OUTPUT
	desideredState: type_LuxGeolumenStatus;
	toSendSetString:STRING;
	toSendGetString:STRING;
END_VAR
VAR
	fltNodeDisappeared:FLT_EVENT;
	retryDisappear:BYTE:=0;
	retryStatusNotAligned:BYTE:=0;
	timerAlive:TON;
	fltNodeStatusNotAligned:FLT_EVENT;
	timerAlignStatus:TON;
	templateDimm : STRING;
	templateGet : STRING;
	tmpNum:STRING;
	commandString:STRING;
	sendString:STRING;
	normalizedDesideredDimmValueGeoLumen:REAL;
	i:INT;
	fNormValue:INT;
END_VAR
;
END_FUNCTION_BLOCK
ACTION checkAlignStatus:
timerAlignStatus(IN:=NOT timerAlignStatus.Q,PT:=T#10s);
IF TimerAlive.Q THEN
	SendDataQueue(pTxData:=ADR(toSendSetString));
	SendDataQueue.addMessage();
	SendDataQueue(pTxData:=ADR(toSendGetString));
	SendDataQueue.addMessage();
	SendDataQueue();
	retryStatusNotAligned:=retryStatusNotAligned+1;
END_IF
END_ACTION
ACTION checkAlive:
TimerAlive(IN:=NOT TimerAlive.Q,PT:=T#3m);
IF TimerAlive.Q THEN
	SendDataQueue(pTxData:=ADR(toSendGetString),ReceiveBufferPtr:=ADR(ReceiveBuffer));
	SendDataQueue.addMessage();
	SendDataQueue();
	retryDisappear:=retryDisappear+1;
END_IF
END_ACTION
ACTION checkStatusANDPresence:
IF(Sys.Time_CT_DT-lastSeen>MAX_NO_FEEDBACK_TIME) AND retryDisappear<MAX_RETRY_NO_FEEDBACK THEN
	checkAlive();
END_IF

fltNodeDisappeared(IN:=(Sys.Time_CT_DT-lastSeen>MAX_NO_FEEDBACK_TIME) AND retryDisappear>=MAX_RETRY_NO_FEEDBACK);
IF fltNodeDisappeared.EVH THEN
	LogEv(EL_Alarm,EO_LUX,ID_Lux,9,'Geolumen node disappeared');
END_IF
IF fltNodeDisappeared.EVL THEN
	LogEv(EL_Alarm,EO_LUX,ID_Lux,1,'Geolumen node came back');
	retryDisappear:=0;
END_IF

IF((isGeolumenIEqualStatus(desideredState,feedbackState)=FALSE) AND retryStatusNotAligned<MAX_RETRY_STATUS_NOT_ALIGNED) THEN
	checkAlignStatus();
END_IF

fltNodeStatusNotAligned(IN:=(isGeolumenIEqualStatus(desideredState,feedbackState)=FALSE)  AND retryStatusNotAligned>=MAX_RETRY_STATUS_NOT_ALIGNED);
IF fltNodeStatusNotAligned.EVH THEN
	LogEv(EL_Alarm,EO_LUX,ID_Lux,9,'Geolumen node with desidered status DIFFERENT from feedback status');
END_IF
IF fltNodeStatusNotAligned.EVL THEN
	LogEv(EL_Alarm,EO_LUX,ID_Lux,1,'Geolumen node with desidered status = feedback status');
	 retryStatusNotAligned:=0;
END_IF
END_ACTION
ACTION updateDesideredState:
desideredState.id_Geolumen:=ID_Geolumen;
normalizedDesideredDimmValueGeoLumen:=(WORD_TO_REAL(desideredDimmValue)/WORD_TO_REAL(MAX_DIMM_LUX_CLEVERGY))*MAX_DIMM;
desideredState.DimmValue_0:=REAL_TO_WORD(normalizedDesideredDimmValueGeoLumen);
desideredState.DimmValue_1:=REAL_TO_WORD(normalizedDesideredDimmValueGeoLumen);
desideredState.DimmValue_2:=REAL_TO_WORD(normalizedDesideredDimmValueGeoLumen);

templateDimm:=',x,x,x$R$N';
tmpNum:=WORD_TO_STRING(REAL_TO_WORD(normalizedDesideredDimmValueGeoLumen));
commandString:=REPLACE_ALL(templateDimm,'x',tmpNum);
sendString := 'NDE_SET_LIGHT=';
sendString:=CONCAT(SendString, DWORD_TO_STRING(ID_Geolumen));
sendString:=CONCAT(SendString, commandString);
toSendSetString:=sendString;
templateGet:='NDE_GET_STATUS=x$R$N';
toSendGetString:=REPLACE_ALL(templateGet,'x',DWORD_TO_STRING(ID_Geolumen));
END_ACTION
ACTION updateFeedbackState:
lastSeen:=Sys.Time_CT_DT;
retryDisappear:=0;
retryStatusNotAligned:=0;
fNormValue:=REAL_TO_INT((WORD_TO_REAL(feedbackState.DimmValue_0)/WORD_TO_REAL(MAX_DIMM))*WORD_TO_REAL(MAX_DIMM_LUX_CLEVERGY));
FOR i:=1 TO MAX_LUXNUM DO
	IF LuxElement[i].ID=ID_Lux THEN
		LuxElement[i](Lux_State:=(fNormValue>0),
		Lux_StateAnalog:=fNormValue,
		WorkingTime:=GlobalWorkingtime[i],
		PowerOnCycles:=GlobalPowerOnCycles[i],
		EnergyCounter:=GlobalEnergyCounter[i],
		EnergyCounter_t:=GlobalEnergyCounter_t[i],KeyQty:=2);
	END_IF
END_FOR
END_ACTION

(* POU objAstroLog, ST *)
FUNCTION objAstroLog:BOOL
VAR_INPUT
	partenza:WORD;
END_VAR
VAR
	groupSize: WORD:=10; (*FACTOR OF GROUPING*)
	groupNumber : WORD;
	i : WORD;
	j : WORD;
	index:WORD;
	isObj : BOOL;
	lastGroup:WORD:=0;
END_VAR
i:=partenza-1;
	(*verifico se nel gruppo corrente c'è qualche ASTR valido *)
	isObj:=FALSE;
	FOR j:=1 TO 10 DO
		index:=i*10+j;
		IF(index<>0 AND index<=MAX_LUXNUM AND ASTR[index].ID<>0 ) THEN isObj:=TRUE; j:=groupSize; END_IF
	END_FOR
	(* se c'è qualche ASTR valido da fare, procedo *)
	IF(isObj) THEN
		Logger_Head();FOR j:=1 TO 10 DO
		index:=i*10+j;
			IF(index<>0 AND index<=MAX_LUXNUM AND ASTR[index].ID<>0 ) THEN ASTR[index].AddLogData(); END_IF
		END_FOR
		Logger_Send();
	END_IF
(*END_FOR*)
END_FUNCTION

(* POU objLuxLog, ST *)
FUNCTION objLuxLog:BOOL
VAR_INPUT
	partenza:WORD;
END_VAR
VAR
	groupSize: WORD:=10; (*FACTOR OF GROUPING*)
	groupNumber : WORD;
	i : WORD;
	j : WORD;
	index:WORD;
	isObj : BOOL;
	lastGroup:WORD:=0;
END_VAR
i:=partenza-1;
	(*verifico se nel gruppo corrente c'è qualche ASTR valido *)
	isObj:=FALSE;
	FOR j:=1 TO 10 DO
		index:=i*10+j;
		IF(index<>0 AND index<=MAX_LUXNUM AND LuxElement[index].ID<>0 ) THEN isObj:=TRUE; j:=groupSize; END_IF
	END_FOR
	(* se c'è qualche ASTR valido da fare, procedo *)
	IF(isObj) THEN
		Logger_Head();FOR j:=1 TO 10 DO
		index:=i*10+j;
			IF(index<>0 AND index<=MAX_LUXNUM AND LuxElement[index].ID<>0 ) THEN

LuxElement[index].AddLogData(WORKINGTIME:=GlobalWorkingtime	[index],
									    POWERONCYCLES:=GlobalPowerOnCycles[index],
									    ENERGYCOUNTER:=GlobalEnergyCounter[index],
									    ENERGYCOUNTER_t :=GlobalEnergyCounter_t[index]);

			END_IF
		END_FOR
		Logger_Send();
	END_IF
(*END_FOR*)
END_FUNCTION

(* POU PLANTCONFIG/Plant_LogTrig, ST *)
FUNCTION Plant_LogTrig : BOOL
VAR_INPUT
END_VAR
VAR
	i:INT;
END_VAR
SyncLogRequest:=TRUE;
timingLuxBase:=t#0m;
timingAstroBase:=t#1m30s;
logRowLux:=0;
logRowAstro:=0;

FOR i:=1 TO 15 DO

TimerLogAstroSyncDone[I]:=FALSE;
TimerLogLuxSyncDone[I]:=FALSE;

END_FOR
END_FUNCTION

(* POU GeoLumenWrapping/SendDataQueue, ST *)
FUNCTION_BLOCK SendDataQueue
VAR CONSTANT
	QUEUE_SIZE:WORD:=1000;
END_VAR
VAR_INPUT
	pTxData: POINTER TO STRING;
	ReceiveBufferPtr : POINTER TO typRing_Buffer;
END_VAR
VAR
	Timer: TON;
	toBeSent : WORD:=0;
	writeIndex:WORD:=0;
	readIndex:WORD:=0;
	StrToSend		: STRING;
	xOpenPort		: BOOL := TRUE;
	xInitPort			: BOOL;
	xStartSend		: BOOL;
	xSendActive	: BOOL;
	xSendActive2	: BOOL;

	pRecStr 	: POINTER TO STRING(255);
	StringFromCom 	: STRING(255);
	tmpStringa : STRING(255) := '';
	LastMsg: STRING(255) := '';

	queue: ARRAY[1..QUEUE_SIZE] OF STRING(255);

	intStart, x : INT;
	counterFrame : INT :=0;
END_VAR
Timer(IN:=NOT Timer.Q,PT:=T#500ms);
IF(Timer.Q AND toBeSent >0) THEN

	readIndex:=((readIndex+1) MOD (QUEUE_SIZE+1))+(readIndex+1)/(QUEUE_SIZE+1);

	StrToSend:=queue[readIndex];
	xSendActive2:= TRUE;

	COM0(	utRECEIVE_BUFFER := ReceiveBufferPtr^,
		ptSEND_BUFFER	:= ADR(StrToSend),
		xINIT				:=  xInitPort,
     		xOPEN_COM_PORT 	:= xOpenPort,
		iBYTES_TO_SEND	:= LEN(StrToSend)+1,
		xSTART_SEND		:= xSendActive2);


	toBeSent:=toBeSent-1;
END_IF
END_FUNCTION_BLOCK
ACTION addMessage:
writeIndex:=((writeIndex+1) MOD (QUEUE_SIZE+1))+(writeIndex+1)/(QUEUE_SIZE+1);

queue[writeIndex]:=pTxData^;

toBeSent:=toBeSent+1;
END_ACTION

(* Visualisation checkNodes
3 elements of other kinds (tables, trends, ...) not read
*)

(* Visualisation CMD_diagn
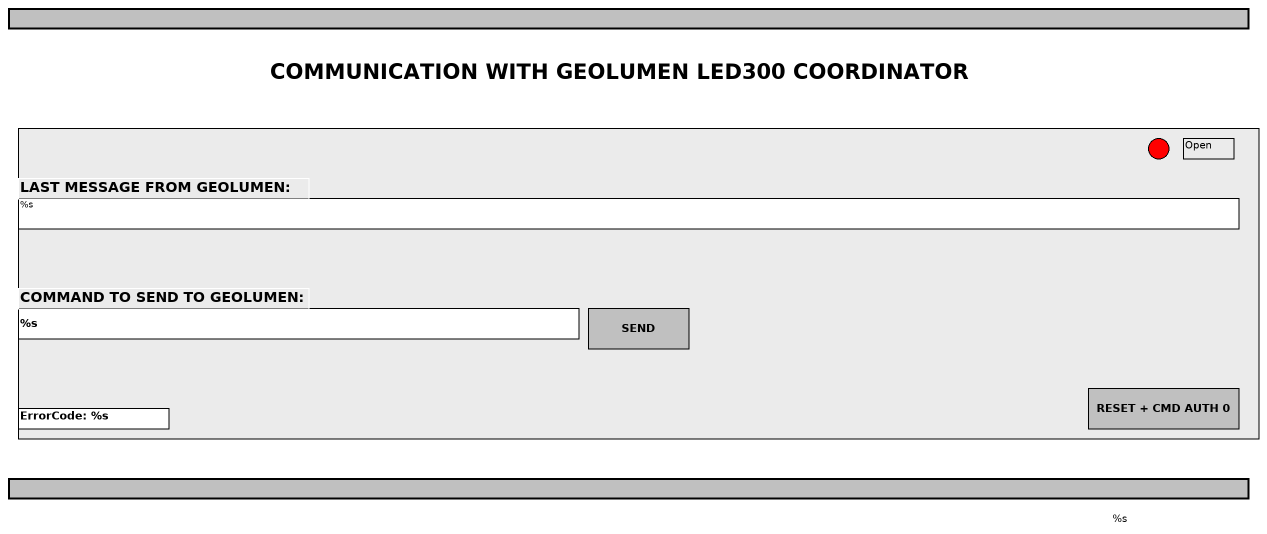
rectangle at (790,500)-(1131,521): text "%s"; shows Sys.Time_LogString
rectangle at (590,300)-(691,341): text "SEND"; runs INTERN ASSIGN LuxGeolumenDiagnostics.executeCommandRequest:=(TRUE)
rectangle at (270,50)-(971,81): text "COMMUNICATION WITH GEOLUMEN LED300 COORDINATOR"
rectangle at (20,300)-(581,331): text "%s"; shows LuxGeolumenDiagnostics.diagnosticCommand; editable
rectangle at (20,190)-(1241,221): text "%s"; shows obj_GeolumenCoordinator.LastMessage
rectangle at (20,400)-(171,421): text "ErrorCode: %s"; shows COM0.bError
rectangle at (1185,130)-(1236,151): text "Open"
ellipse at (1150,130)-(1171,151): alarm colour if COM0.COM_PORT_IST_OFFEN
rectangle at (20,170)-(311,191): text "LAST MESSAGE FROM GEOLUMEN:"
rectangle at (20,280)-(311,301): text "COMMAND TO SEND TO GEOLUMEN:"
rectangle at (1090,380)-(1241,421): text "RESET + CMD AUTH 0"; runs INTERN ASSIGN LuxGeolumenDiagnostics.executeCommandResetRequest:=(TRUE)
3 more shapes without text or variables
*)

(* Visualisation Light_Test
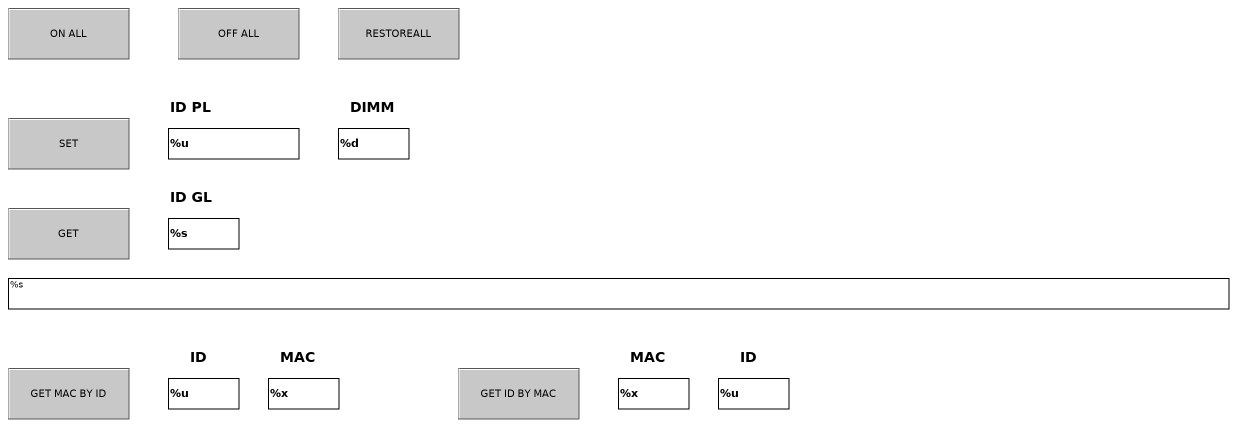
button at (20,10)-(141,61): text "ON ALL"; runs INTERN ASSIGN LuxGeolumenDiagnostics.turnOnRequest:=(TRUE)
button at (190,10)-(311,61): text "OFF ALL"; runs INTERN ASSIGN LuxGeolumenDiagnostics.turnOffRequest:=(TRUE)
button at (20,120)-(141,171): text "SET"; runs INTERN ASSIGN LuxGeolumenDiagnostics.executeCommandSetRequest:=(TRUE)
rectangle at (180,130)-(311,161): text "%u"; shows LuxGeolumenDiagnostics.commandSetID; editable
rectangle at (350,130)-(421,161): text "%d"; shows LuxGeolumenDiagnostics.commandSetDIMM; editable
rectangle at (180,100)-(231,121): text "ID PL"
rectangle at (360,100)-(411,121): text "DIMM"
button at (20,210)-(141,261): text "GET"; runs INTERN ASSIGN LuxGeolumenDiagnostics.executeCommandGetRequest:=(TRUE)
rectangle at (180,220)-(251,251): text "%s"; shows LuxGeolumenDiagnostics.commandGetID; editable
rectangle at (180,190)-(241,211): text "ID GL"
rectangle at (20,280)-(1241,311): text "%s"; shows obj_GeolumenCoordinator.LastMessage
button at (20,370)-(141,421): text "GET MAC BY ID"; runs INTERN ASSIGN LuxGeolumenDiagnostics.executeCommandGetMACByIDRequest:=(TRUE)
rectangle at (180,380)-(251,411): text "%u"; shows LuxGeolumenDiagnostics.commandGetMacByID; editable
rectangle at (280,380)-(351,411): text "%x"; shows LuxGeolumenDiagnostics.commandGetMacByIDResult; editable
rectangle at (200,350)-(231,371): text "ID"
rectangle at (290,350)-(341,371): text "MAC"
button at (470,370)-(591,421): text "GET ID BY MAC"; runs INTERN ASSIGN LuxGeolumenDiagnostics.executeCommandGetIDByMACRequest:=(TRUE)
rectangle at (730,380)-(801,411): text "%u"; shows LuxGeolumenDiagnostics.commandGetIDByMacResult; editable
rectangle at (630,380)-(701,411): text "%x"; shows LuxGeolumenDiagnostics.commandGetIDByMac; editable
rectangle at (750,350)-(781,371): text "ID"
rectangle at (640,350)-(691,371): text "MAC"
button at (350,10)-(471,61): text "RESTOREALL"; runs INTERN ASSIGN LuxGeolumenDiagnostics.restoreAllRequest:=(TRUE)
*)

(* Visualisation LUX_Status
1 elements of other kinds (tables, trends, ...) not read
*)

(* Visualisation PLC_VISU
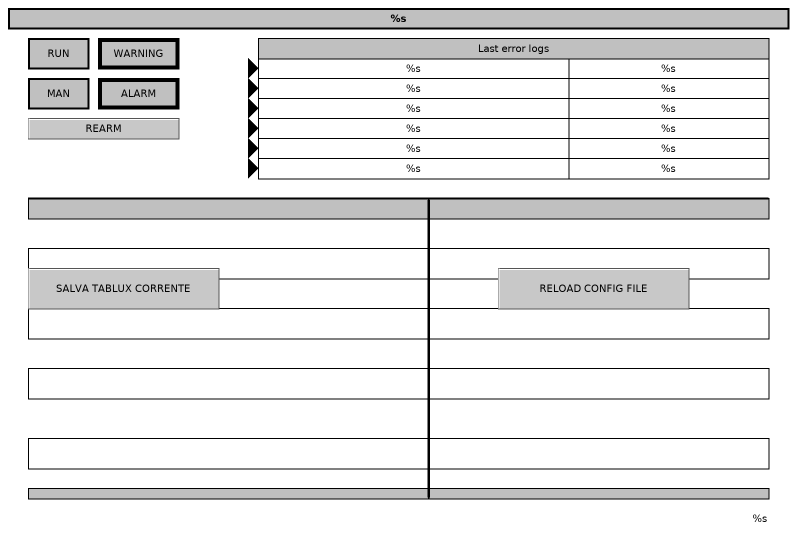
rectangle at (10,0)-(791,21): text "%s"; shows .Plant_NAME
rounded rectangle at (30,30)-(91,61): text "RUN"; alarm colour if NOT Mode_Manual; runs INTERN ASSIGN Mode_Manual:=(FALSE)
rounded rectangle at (30,70)-(91,101): text "MAN"; alarm colour if Mode_Manual; runs INTERN ASSIGN Mode_Manual:=(TRUE)
rectangle at (570,50)-(771,71): text "%s"; shows Sys.LastLogs_Msg[0]
polygon at (250,150)-(260,170): invisible if Sys.LastLogs_Idx<>0
rectangle at (570,70)-(771,91): text "%s"; shows Sys.LastLogs_Msg[1]
polygon at (250,50)-(260,70): invisible if Sys.LastLogs_Idx<>1
rectangle at (570,90)-(771,111): text "%s"; shows Sys.LastLogs_Msg[2]
polygon at (250,70)-(260,90): invisible if Sys.LastLogs_Idx<>2
rectangle at (570,110)-(771,131): text "%s"; shows Sys.LastLogs_Msg[3]
polygon at (250,90)-(260,110): invisible if Sys.LastLogs_Idx<>3
rectangle at (570,130)-(771,151): text "%s"; shows Sys.LastLogs_Msg[4]
polygon at (250,110)-(260,130): invisible if Sys.LastLogs_Idx<>4
rectangle at (570,150)-(771,171): text "%s"; shows Sys.LastLogs_Msg[5]
polygon at (250,130)-(260,150): invisible if Sys.LastLogs_Idx<>5
rectangle at (260,50)-(571,71): text "%s"; shows Sys.LastLogs_Dat[0]
rectangle at (260,70)-(571,91): text "%s"; shows Sys.LastLogs_Dat[1]
rectangle at (260,90)-(571,111): text "%s"; shows Sys.LastLogs_Dat[2]
rectangle at (260,110)-(571,131): text "%s"; shows Sys.LastLogs_Dat[3]
rectangle at (260,130)-(571,151): text "%s"; shows Sys.LastLogs_Dat[4]
rectangle at (260,150)-(571,171): text "%s"; shows Sys.LastLogs_Dat[5]
rectangle at (100,70)-(181,101): text "ALARM"; alarm colour if Sys.Alarm; runs INTERN ASSIGN Mode_Manual:=(FALSE)
rectangle at (100,30)-(181,61): text "WARNING"; alarm colour if Sys.Warning; runs INTERN ASSIGN Mode_Manual:=(TRUE)
button at (30,110)-(181,131): text "REARM"; runs INTERN ASSIGN Sys.Alarm:=(FALSE);INTERN ASSIGN Sys.Warning:=(FALSE)
rectangle at (260,30)-(771,51): text "Last error logs"
rectangle at (430,500)-(771,521): text "%s"; shows Sys.Time_LogString
button at (30,260)-(221,301): text "SALVA TABLUX CORRENTE"; runs INTERN ASSIGN LuxGeolumenDiagnostics.executeCommandSaveToFileRequest:=(TRUE)
button at (500,260)-(691,301): text "RELOAD CONFIG FILE"; runs INTERN ASSIGN Sys.Status:=(S_RELOAD)
8 more shapes without text or variables
*)

